(* Logix 5000 project; controller LeakTestAuto vendor 1 type 14 code 226 rev 37.11; software revision 37.01; part 7 of 15 *)
(* tags used below, declared in another part *)
   ConveyorPurgeCounter : DINT;   // Outfeed Coveyor Purge Counter
   DateString : String20;
   DateTimeString : String20;
   HMI_PurgeCycleSP : DINT;   // HMI Purge Cycles Setpoint
   I_OP220_N3_CONVEYOR_CLEAT : ALIAS FOR Local:3:I.Pt13.Data;
   I_OP220_N3_CONVEYOR_LOAD : ALIAS FOR Local:3:I.Pt12.Data;
   I_OP220_N3_CONVEYOR_UNLOAD : ALIAS FOR Local:3:I.Pt14.Data;
   I_OP220_N3_DUT_PRE_NEST_0 : ALIAS FOR Local:3:I.Pt00.Data;
   I_OP220_N3_DUT_PRE_NEST_1 : ALIAS FOR Local:3:I.Pt01.Data;
   I_OP220_N3_DUT_PRE_NEST_2 : ALIAS FOR Local:3:I.Pt02.Data;
   I_OP220_N3_MAIN_AIR_OK : ALIAS FOR Local:3:I.Pt07.Data;
   I_OP220_N3_NEST1_EXTEND : ALIAS FOR Local:3:I.Pt04.Data;
   I_OP220_N3_NEST1_HOME : ALIAS FOR Local:3:I.Pt03.Data;
   I_OP220_N3_NEST2_EXTEND : ALIAS FOR Local:3:I.Pt06.Data;
   I_OP220_N3_NEST2_HOME : ALIAS FOR Local:3:I.Pt05.Data;
   I_OP220_N3_REJECT_BIN_OK : ALIAS FOR Local:3:I.Pt09.Data;
   IOCounterHasRef : BOOL;
   IOTriggerCounts : UDINT[128];
   James_Dint : DINT;   // James Test Word
   LastPLCEdit : String20;
   LastPLCEditHistory : String20[20];
   O_OP220_N5_EN_LT_BU : ALIAS FOR Local:5:O.Pt03.Data;
   O_OP220_N5_EN_LT_GN : ALIAS FOR Local:5:O.Pt00.Data;
   O_OP220_N5_EN_LT_RD : ALIAS FOR Local:5:O.Pt02.Data;
   O_OP220_N5_EN_LT_YE : ALIAS FOR Local:5:O.Pt01.Data;
   OP220_ConsumedFromMain_PurgeModeEn : BOOL;
   OP220_Power : BOOL;
   PLC : AOI_PLC;
   Purge_Count_DN : BOOL;   // Purge Counter Completed
   ShiftChange : BOOL;
   ShiftNumber : SINT;
   TimeString : String20;
   TON_PLC_BootUp : TIMER;

        [95].VolumeTest.Detailed.Test_Type := 69, [95].VolumeTest.Detailed.element_data[0].Variable_code := 245, [95].VolumeTest.Detailed.element_data[0].prec_code := 2, [95].VolumeTest.Detailed.element_data[0].Unit_code := 165, [95].VolumeTest.Detailed.element_data[0].result_measurement := 188.38309, [95].VolumeTest.Detailed.element_data[1].Variable_code := 13, [95].VolumeTest.Detailed.element_data[1].prec_code := 3, [95].VolumeTest.Detailed.element_data[1].Unit_code := 12, [95].VolumeTest.Detailed.element_data[1].result_measurement := 1.8068217, [95].VolumeTest.Detailed.element_data[2].Variable_code := 247, [95].VolumeTest.Detailed.element_data[2].prec_code := 3, [95].VolumeTest.Detailed.element_data[2].Unit_code := 12, [95].VolumeTest.Detailed.element_data[2].result_measurement := 5.2105684, [95].VolumeTest.Detailed.element_data[3].Variable_code := 295, [95].VolumeTest.Detailed.element_data[3].prec_code := 3, [95].VolumeTest.Detailed.element_data[3].Unit_code := 12, [95].VolumeTest.Detailed.element_data[3].result_measurement := 5.212333, [95].LeakTest.UID := 42962, [95].LeakTest.Basic.unique_id := 42962, [95].LeakTest.Basic.channel_num := 1, [95].LeakTest.Basic.program_num := 2, [95].LeakTest.Basic.evaluation_code := 1, [95].LeakTest.Basic.test_port := 1, [95].LeakTest.Basic.year := 26, [95].LeakTest.Basic.month := 6, [95].LeakTest.Basic.date := 4, [95].LeakTest.Basic.hour := 15, [95].LeakTest.Basic.minute := 9, [95].LeakTest.Basic.second := 47, [95].LeakTest.Basic.flags := 12, [95].LeakTest.Basic.Num_tests := 1, [95].LeakTest.Basic.test_elements.test_type := 66, [95].LeakTest.Basic.test_elements.test_eval := 1, [95].LeakTest.Basic.test_elements.num_elements := 16, [95].LeakTest.Detailed.unique_id := 42962, [95].LeakTest.Detailed.num_elements := 16, [95].LeakTest.Detailed.Test_Type := 66, [95].LeakTest.Detailed.element_data[0].Variable_code := 61, [95].LeakTest.Detailed.element_data[0].prec_code := 2, [95].LeakTest.Detailed.element_data[0].Unit_code := 60, [95].LeakTest.Detailed.element_data[0].result_measurement := 0.022351742, [95].LeakTest.Detailed.element_data[1].Variable_code := 28, [95].LeakTest.Detailed.element_data[1].prec_code := 3, [95].LeakTest.Detailed.element_data[1].Unit_code := 41, [95].LeakTest.Detailed.element_data[1].result_measurement := 0.0004656613, [95].LeakTest.Detailed.element_data[2].Variable_code := 13, [95].LeakTest.Detailed.element_data[2].prec_code := 3, [95].LeakTest.Detailed.element_data[2].Unit_code := 12, [95].LeakTest.Detailed.element_data[2].result_measurement := 5.2300653, [95].LeakTest.Detailed.element_data[3].Variable_code := 75, [95].LeakTest.Detailed.element_data[3].prec_code := 2, [95].LeakTest.Detailed.element_data[3].Unit_code := 60, [95].LeakTest.Detailed.element_data[4].Variable_code := 60, [95].LeakTest.Detailed.element_data[4].prec_code := 2, [95].LeakTest.Detailed.element_data[4].Unit_code := 60, [95].LeakTest.Detailed.element_data[4].result_measurement := 0.022910535, [95].LeakTest.Detailed.element_data[5].Variable_code := 56, [95].LeakTest.Detailed.element_data[5].prec_code := 3, [95].LeakTest.Detailed.element_data[5].Unit_code := 41, [95].LeakTest.Detailed.element_data[5].result_measurement := 0.00020023435,
        [95].LeakTest.Detailed.element_data[6].Variable_code := 55, [95].LeakTest.Detailed.element_data[6].prec_code := 3, [95].LeakTest.Detailed.element_data[6].Unit_code := 12, [95].LeakTest.Detailed.element_data[6].result_measurement := 5.2300653, [95].LeakTest.Detailed.element_data[7].Variable_code := 58, [95].LeakTest.Detailed.element_data[7].prec_code := 2, [95].LeakTest.Detailed.element_data[7].Unit_code := 60, [95].LeakTest.Detailed.element_data[7].result_measurement := -1.0002404, [95].LeakTest.Detailed.element_data[8].Variable_code := 59, [95].LeakTest.Detailed.element_data[8].prec_code := 2, [95].LeakTest.Detailed.element_data[8].Unit_code := 60, [95].LeakTest.Detailed.element_data[8].result_measurement := 1.0002404, [95].LeakTest.Detailed.element_data[9].Variable_code := 12, [95].LeakTest.Detailed.element_data[9].prec_code := 3, [95].LeakTest.Detailed.element_data[9].Unit_code := 12, [95].LeakTest.Detailed.element_data[9].result_measurement := 5.000001, [95].LeakTest.Detailed.element_data[10].Variable_code := 62, [95].LeakTest.Detailed.element_data[10].prec_code := 2, [95].LeakTest.Detailed.element_data[10].Unit_code := 60, [95].LeakTest.Detailed.element_data[10].result_measurement := 1.1298805, [95].LeakTest.Detailed.element_data[11].Variable_code := 21, [95].LeakTest.Detailed.element_data[11].prec_code := 3, [95].LeakTest.Detailed.element_data[11].Unit_code := 41, [95].LeakTest.Detailed.element_data[11].result_measurement := 4.656613e-06, [95].LeakTest.Detailed.element_data[12].Variable_code := 25, [95].LeakTest.Detailed.element_data[12].prec_code := 3, [95].LeakTest.Detailed.element_data[12].Unit_code := 41, [95].LeakTest.Detailed.element_data[12].result_measurement := 0.023245811, [95].LeakTest.Detailed.element_data[13].Variable_code := 216, [95].LeakTest.Detailed.element_data[13].prec_code := 3, [95].LeakTest.Detailed.element_data[13].Unit_code := 41, [95].LeakTest.Detailed.element_data[13].result_measurement := -3.7252903e-05, [95].LeakTest.Detailed.element_data[14].Variable_code := 218, [95].LeakTest.Detailed.element_data[14].prec_code := 3, [95].LeakTest.Detailed.element_data[14].Unit_code := 41, [95].LeakTest.Detailed.element_data[14].result_measurement := 0.011632219, [95].LeakTest.Detailed.element_data[15].Variable_code := 295, [95].LeakTest.Detailed.element_data[15].prec_code := 3, [95].LeakTest.Detailed.element_data[15].Unit_code := 12, [95].LeakTest.Detailed.element_data[15].result_measurement := 5.231574, [96].Barcode := 'B252620865', [96].VolumeTest.UID := 42009, [96].VolumeTest.Basic.unique_id := 42009, [96].VolumeTest.Basic.channel_num := 1, [96].VolumeTest.Basic.program_num := 1, [96].VolumeTest.Basic.evaluation_code := 1, [96].VolumeTest.Basic.test_port := 1, [96].VolumeTest.Basic.year := 26, [96].VolumeTest.Basic.month := 6, [96].VolumeTest.Basic.date := 5, [96].VolumeTest.Basic.hour := 10, [96].VolumeTest.Basic.minute := 13, [96].VolumeTest.Basic.second := 35, [96].VolumeTest.Basic.flags := 12, [96].VolumeTest.Basic.Num_tests := 1, [96].VolumeTest.Basic.test_elements.test_type := 69, [96].VolumeTest.Basic.test_elements.test_eval := 1, [96].VolumeTest.Basic.test_elements.num_elements := 4, [96].VolumeTest.Detailed.unique_id := 42009, [96].VolumeTest.Detailed.num_elements := 4,
        [96].VolumeTest.Detailed.Test_Type := 69, [96].VolumeTest.Detailed.element_data[0].Variable_code := 245, [96].VolumeTest.Detailed.element_data[0].prec_code := 2, [96].VolumeTest.Detailed.element_data[0].Unit_code := 165, [96].VolumeTest.Detailed.element_data[0].result_measurement := 185.74803, [96].VolumeTest.Detailed.element_data[1].Variable_code := 13, [96].VolumeTest.Detailed.element_data[1].prec_code := 3, [96].VolumeTest.Detailed.element_data[1].Unit_code := 12, [96].VolumeTest.Detailed.element_data[1].result_measurement := 1.7781556, [96].VolumeTest.Detailed.element_data[2].Variable_code := 247, [96].VolumeTest.Detailed.element_data[2].prec_code := 3, [96].VolumeTest.Detailed.element_data[2].Unit_code := 12, [96].VolumeTest.Detailed.element_data[2].result_measurement := 5.0810447, [96].VolumeTest.Detailed.element_data[3].Variable_code := 295, [96].VolumeTest.Detailed.element_data[3].prec_code := 3, [96].VolumeTest.Detailed.element_data[3].Unit_code := 12, [96].VolumeTest.Detailed.element_data[3].result_measurement := 5.081105, [96].LeakTest.UID := 42010, [96].LeakTest.Basic.unique_id := 42010, [96].LeakTest.Basic.channel_num := 1, [96].LeakTest.Basic.program_num := 2, [96].LeakTest.Basic.evaluation_code := 1, [96].LeakTest.Basic.test_port := 1, [96].LeakTest.Basic.year := 26, [96].LeakTest.Basic.month := 6, [96].LeakTest.Basic.date := 5, [96].LeakTest.Basic.hour := 10, [96].LeakTest.Basic.minute := 13, [96].LeakTest.Basic.second := 42, [96].LeakTest.Basic.flags := 12, [96].LeakTest.Basic.Num_tests := 1, [96].LeakTest.Basic.test_elements.test_type := 66, [96].LeakTest.Basic.test_elements.test_eval := 1, [96].LeakTest.Basic.test_elements.num_elements := 16, [96].LeakTest.Detailed.unique_id := 42010, [96].LeakTest.Detailed.num_elements := 16, [96].LeakTest.Detailed.Test_Type := 66, [96].LeakTest.Detailed.element_data[0].Variable_code := 61, [96].LeakTest.Detailed.element_data[0].prec_code := 2, [96].LeakTest.Detailed.element_data[0].Unit_code := 60, [96].LeakTest.Detailed.element_data[0].result_measurement := -0.067055225, [96].LeakTest.Detailed.element_data[1].Variable_code := 28, [96].LeakTest.Detailed.element_data[1].prec_code := 3, [96].LeakTest.Detailed.element_data[1].Unit_code := 41, [96].LeakTest.Detailed.element_data[1].result_measurement := 0.00027939677, [96].LeakTest.Detailed.element_data[2].Variable_code := 13, [96].LeakTest.Detailed.element_data[2].prec_code := 3, [96].LeakTest.Detailed.element_data[2].Unit_code := 12, [96].LeakTest.Detailed.element_data[2].result_measurement := 5.1023254, [96].LeakTest.Detailed.element_data[3].Variable_code := 75, [96].LeakTest.Detailed.element_data[3].prec_code := 2, [96].LeakTest.Detailed.element_data[3].Unit_code := 60, [96].LeakTest.Detailed.element_data[4].Variable_code := 60, [96].LeakTest.Detailed.element_data[4].prec_code := 2, [96].LeakTest.Detailed.element_data[4].Unit_code := 60, [96].LeakTest.Detailed.element_data[4].result_measurement := -0.07208437, [96].LeakTest.Detailed.element_data[5].Variable_code := 56, [96].LeakTest.Detailed.element_data[5].prec_code := 3, [96].LeakTest.Detailed.element_data[5].Unit_code := 41, [96].LeakTest.Detailed.element_data[5].result_measurement := 0.00019092113,
        [96].LeakTest.Detailed.element_data[6].Variable_code := 55, [96].LeakTest.Detailed.element_data[6].prec_code := 3, [96].LeakTest.Detailed.element_data[6].Unit_code := 12, [96].LeakTest.Detailed.element_data[6].result_measurement := 5.1023254, [96].LeakTest.Detailed.element_data[7].Variable_code := 58, [96].LeakTest.Detailed.element_data[7].prec_code := 2, [96].LeakTest.Detailed.element_data[7].Unit_code := 60, [96].LeakTest.Detailed.element_data[7].result_measurement := -1.0002404, [96].LeakTest.Detailed.element_data[8].Variable_code := 59, [96].LeakTest.Detailed.element_data[8].prec_code := 2, [96].LeakTest.Detailed.element_data[8].Unit_code := 60, [96].LeakTest.Detailed.element_data[8].result_measurement := 1.0002404, [96].LeakTest.Detailed.element_data[9].Variable_code := 12, [96].LeakTest.Detailed.element_data[9].prec_code := 3, [96].LeakTest.Detailed.element_data[9].Unit_code := 12, [96].LeakTest.Detailed.element_data[9].result_measurement := 5.000001, [96].LeakTest.Detailed.element_data[10].Variable_code := 62, [96].LeakTest.Detailed.element_data[10].prec_code := 2, [96].LeakTest.Detailed.element_data[10].Unit_code := 60, [96].LeakTest.Detailed.element_data[10].result_measurement := 1.1002644, [96].LeakTest.Detailed.element_data[11].Variable_code := 21, [96].LeakTest.Detailed.element_data[11].prec_code := 3, [96].LeakTest.Detailed.element_data[11].Unit_code := 41, [96].LeakTest.Detailed.element_data[11].result_measurement := 0.0015180558, [96].LeakTest.Detailed.element_data[12].Variable_code := 25, [96].LeakTest.Detailed.element_data[12].prec_code := 3, [96].LeakTest.Detailed.element_data[12].Unit_code := 41, [96].LeakTest.Detailed.element_data[12].result_measurement := 0.021727756, [96].LeakTest.Detailed.element_data[13].Variable_code := 216, [96].LeakTest.Detailed.element_data[13].prec_code := 3, [96].LeakTest.Detailed.element_data[13].Unit_code := 41, [96].LeakTest.Detailed.element_data[13].result_measurement := 0.00085681677, [96].LeakTest.Detailed.element_data[14].Variable_code := 218, [96].LeakTest.Detailed.element_data[14].prec_code := 3, [96].LeakTest.Detailed.element_data[14].Unit_code := 41, [96].LeakTest.Detailed.element_data[14].result_measurement := 0.01094304, [96].LeakTest.Detailed.element_data[15].Variable_code := 295, [96].LeakTest.Detailed.element_data[15].prec_code := 3, [96].LeakTest.Detailed.element_data[15].Unit_code := 12, [96].LeakTest.Detailed.element_data[15].result_measurement := 5.1039925, [97].Barcode := 'B252620970', [97].VolumeTest.UID := 42015, [97].VolumeTest.Basic.unique_id := 42015, [97].VolumeTest.Basic.channel_num := 1, [97].VolumeTest.Basic.program_num := 1, [97].VolumeTest.Basic.evaluation_code := 1, [97].VolumeTest.Basic.test_port := 1, [97].VolumeTest.Basic.year := 26, [97].VolumeTest.Basic.month := 6, [97].VolumeTest.Basic.date := 5, [97].VolumeTest.Basic.hour := 10, [97].VolumeTest.Basic.minute := 18, [97].VolumeTest.Basic.second := 26, [97].VolumeTest.Basic.flags := 12, [97].VolumeTest.Basic.Num_tests := 1, [97].VolumeTest.Basic.test_elements.test_type := 69, [97].VolumeTest.Basic.test_elements.test_eval := 1, [97].VolumeTest.Basic.test_elements.num_elements := 4, [97].VolumeTest.Detailed.unique_id := 42015, [97].VolumeTest.Detailed.num_elements := 4,
        [97].VolumeTest.Detailed.Test_Type := 69, [97].VolumeTest.Detailed.element_data[0].Variable_code := 245, [97].VolumeTest.Detailed.element_data[0].prec_code := 2, [97].VolumeTest.Detailed.element_data[0].Unit_code := 165, [97].VolumeTest.Detailed.element_data[0].result_measurement := 185.95625, [97].VolumeTest.Detailed.element_data[1].Variable_code := 13, [97].VolumeTest.Detailed.element_data[1].prec_code := 3, [97].VolumeTest.Detailed.element_data[1].Unit_code := 12, [97].VolumeTest.Detailed.element_data[1].result_measurement := 1.778258, [97].VolumeTest.Detailed.element_data[2].Variable_code := 247, [97].VolumeTest.Detailed.element_data[2].prec_code := 3, [97].VolumeTest.Detailed.element_data[2].Unit_code := 12, [97].VolumeTest.Detailed.element_data[2].result_measurement := 5.08504, [97].VolumeTest.Detailed.element_data[3].Variable_code := 295, [97].VolumeTest.Detailed.element_data[3].prec_code := 3, [97].VolumeTest.Detailed.element_data[3].Unit_code := 12, [97].VolumeTest.Detailed.element_data[3].result_measurement := 5.086218, [97].LeakTest.UID := 42016, [97].LeakTest.Basic.unique_id := 42016, [97].LeakTest.Basic.channel_num := 1, [97].LeakTest.Basic.program_num := 2, [97].LeakTest.Basic.evaluation_code := 1, [97].LeakTest.Basic.test_port := 1, [97].LeakTest.Basic.year := 26, [97].LeakTest.Basic.month := 6, [97].LeakTest.Basic.date := 5, [97].LeakTest.Basic.hour := 10, [97].LeakTest.Basic.minute := 18, [97].LeakTest.Basic.second := 33, [97].LeakTest.Basic.flags := 12, [97].LeakTest.Basic.Num_tests := 1, [97].LeakTest.Basic.test_elements.test_type := 66, [97].LeakTest.Basic.test_elements.test_eval := 1, [97].LeakTest.Basic.test_elements.num_elements := 16, [97].LeakTest.Detailed.unique_id := 42016, [97].LeakTest.Detailed.num_elements := 16, [97].LeakTest.Detailed.Test_Type := 66, [97].LeakTest.Detailed.element_data[0].Variable_code := 61, [97].LeakTest.Detailed.element_data[0].prec_code := 2, [97].LeakTest.Detailed.element_data[0].Unit_code := 60, [97].LeakTest.Detailed.element_data[0].result_measurement := -0.0692904, [97].LeakTest.Detailed.element_data[1].Variable_code := 28, [97].LeakTest.Detailed.element_data[1].prec_code := 3, [97].LeakTest.Detailed.element_data[1].Unit_code := 41, [97].LeakTest.Detailed.element_data[1].result_measurement := 0.00023748726, [97].LeakTest.Detailed.element_data[2].Variable_code := 13, [97].LeakTest.Detailed.element_data[2].prec_code := 3, [97].LeakTest.Detailed.element_data[2].Unit_code := 12, [97].LeakTest.Detailed.element_data[2].result_measurement := 5.1036057, [97].LeakTest.Detailed.element_data[3].Variable_code := 75, [97].LeakTest.Detailed.element_data[3].prec_code := 2, [97].LeakTest.Detailed.element_data[3].Unit_code := 60, [97].LeakTest.Detailed.element_data[4].Variable_code := 60, [97].LeakTest.Detailed.element_data[4].prec_code := 2, [97].LeakTest.Detailed.element_data[4].Unit_code := 60, [97].LeakTest.Detailed.element_data[4].result_measurement := -0.073201954, [97].LeakTest.Detailed.element_data[5].Variable_code := 56, [97].LeakTest.Detailed.element_data[5].prec_code := 3, [97].LeakTest.Detailed.element_data[5].Unit_code := 41, [97].LeakTest.Detailed.element_data[5].result_measurement := 0.0001816079,
        [97].LeakTest.Detailed.element_data[6].Variable_code := 55, [97].LeakTest.Detailed.element_data[6].prec_code := 3, [97].LeakTest.Detailed.element_data[6].Unit_code := 12, [97].LeakTest.Detailed.element_data[6].result_measurement := 5.1036057, [97].LeakTest.Detailed.element_data[7].Variable_code := 58, [97].LeakTest.Detailed.element_data[7].prec_code := 2, [97].LeakTest.Detailed.element_data[7].Unit_code := 60, [97].LeakTest.Detailed.element_data[7].result_measurement := -1.0002404, [97].LeakTest.Detailed.element_data[8].Variable_code := 59, [97].LeakTest.Detailed.element_data[8].prec_code := 2, [97].LeakTest.Detailed.element_data[8].Unit_code := 60, [97].LeakTest.Detailed.element_data[8].result_measurement := 1.0002404, [97].LeakTest.Detailed.element_data[9].Variable_code := 12, [97].LeakTest.Detailed.element_data[9].prec_code := 3, [97].LeakTest.Detailed.element_data[9].Unit_code := 12, [97].LeakTest.Detailed.element_data[9].result_measurement := 5.000001, [97].LeakTest.Detailed.element_data[10].Variable_code := 62, [97].LeakTest.Detailed.element_data[10].prec_code := 2, [97].LeakTest.Detailed.element_data[10].Unit_code := 60, [97].LeakTest.Detailed.element_data[10].result_measurement := 1.1002644, [97].LeakTest.Detailed.element_data[11].Variable_code := 21, [97].LeakTest.Detailed.element_data[11].prec_code := 3, [97].LeakTest.Detailed.element_data[11].Unit_code := 41, [97].LeakTest.Detailed.element_data[11].result_measurement := 0.0015180558, [97].LeakTest.Detailed.element_data[12].Variable_code := 25, [97].LeakTest.Detailed.element_data[12].prec_code := 3, [97].LeakTest.Detailed.element_data[12].Unit_code := 41, [97].LeakTest.Detailed.element_data[12].result_measurement := 0.021727756, [97].LeakTest.Detailed.element_data[13].Variable_code := 216, [97].LeakTest.Detailed.element_data[13].prec_code := 3, [97].LeakTest.Detailed.element_data[13].Unit_code := 41, [97].LeakTest.Detailed.element_data[13].result_measurement := 0.00085681677, [97].LeakTest.Detailed.element_data[14].Variable_code := 218, [97].LeakTest.Detailed.element_data[14].prec_code := 3, [97].LeakTest.Detailed.element_data[14].Unit_code := 41, [97].LeakTest.Detailed.element_data[14].result_measurement := 0.01094304, [97].LeakTest.Detailed.element_data[15].Variable_code := 295, [97].LeakTest.Detailed.element_data[15].prec_code := 3, [97].LeakTest.Detailed.element_data[15].Unit_code := 12, [97].LeakTest.Detailed.element_data[15].result_measurement := 5.1049933, [98].Barcode := 'B252620571', [98].VolumeTest.UID := 43010, [98].VolumeTest.Basic.unique_id := 43010, [98].VolumeTest.Basic.channel_num := 1, [98].VolumeTest.Basic.program_num := 1, [98].VolumeTest.Basic.evaluation_code := 1, [98].VolumeTest.Basic.test_port := 1, [98].VolumeTest.Basic.year := 26, [98].VolumeTest.Basic.month := 6, [98].VolumeTest.Basic.date := 5, [98].VolumeTest.Basic.hour := 10, [98].VolumeTest.Basic.minute := 18, [98].VolumeTest.Basic.second := 50, [98].VolumeTest.Basic.flags := 12, [98].VolumeTest.Basic.Num_tests := 1, [98].VolumeTest.Basic.test_elements.test_type := 69, [98].VolumeTest.Basic.test_elements.test_eval := 1, [98].VolumeTest.Basic.test_elements.num_elements := 4, [98].VolumeTest.Detailed.unique_id := 43010, [98].VolumeTest.Detailed.num_elements := 4,
        [98].VolumeTest.Detailed.Test_Type := 69, [98].VolumeTest.Detailed.element_data[0].Variable_code := 245, [98].VolumeTest.Detailed.element_data[0].prec_code := 2, [98].VolumeTest.Detailed.element_data[0].Unit_code := 165, [98].VolumeTest.Detailed.element_data[0].result_measurement := 187.18771, [98].VolumeTest.Detailed.element_data[1].Variable_code := 13, [98].VolumeTest.Detailed.element_data[1].prec_code := 3, [98].VolumeTest.Detailed.element_data[1].Unit_code := 12, [98].VolumeTest.Detailed.element_data[1].result_measurement := 1.7792639, [98].VolumeTest.Detailed.element_data[2].Variable_code := 247, [98].VolumeTest.Detailed.element_data[2].prec_code := 3, [98].VolumeTest.Detailed.element_data[2].Unit_code := 12, [98].VolumeTest.Detailed.element_data[2].result_measurement := 5.109827, [98].VolumeTest.Detailed.element_data[3].Variable_code := 295, [98].VolumeTest.Detailed.element_data[3].prec_code := 3, [98].VolumeTest.Detailed.element_data[3].Unit_code := 12, [98].VolumeTest.Detailed.element_data[3].result_measurement := 5.1112704, [98].LeakTest.UID := 43011, [98].LeakTest.Basic.unique_id := 43011, [98].LeakTest.Basic.channel_num := 1, [98].LeakTest.Basic.program_num := 2, [98].LeakTest.Basic.evaluation_code := 1, [98].LeakTest.Basic.test_port := 1, [98].LeakTest.Basic.year := 26, [98].LeakTest.Basic.month := 6, [98].LeakTest.Basic.date := 5, [98].LeakTest.Basic.hour := 10, [98].LeakTest.Basic.minute := 18, [98].LeakTest.Basic.second := 57, [98].LeakTest.Basic.flags := 12, [98].LeakTest.Basic.Num_tests := 1, [98].LeakTest.Basic.test_elements.test_type := 66, [98].LeakTest.Basic.test_elements.test_eval := 1, [98].LeakTest.Basic.test_elements.num_elements := 16, [98].LeakTest.Detailed.unique_id := 43011, [98].LeakTest.Detailed.num_elements := 16, [98].LeakTest.Detailed.Test_Type := 66, [98].LeakTest.Detailed.element_data[0].Variable_code := 61, [98].LeakTest.Detailed.element_data[0].prec_code := 2, [98].LeakTest.Detailed.element_data[0].Unit_code := 60, [98].LeakTest.Detailed.element_data[0].result_measurement := -0.0033527613, [98].LeakTest.Detailed.element_data[1].Variable_code := 28, [98].LeakTest.Detailed.element_data[1].prec_code := 3, [98].LeakTest.Detailed.element_data[1].Unit_code := 41, [98].LeakTest.Detailed.element_data[1].result_measurement := -7.4505806e-05, [98].LeakTest.Detailed.element_data[2].Variable_code := 13, [98].LeakTest.Detailed.element_data[2].prec_code := 3, [98].LeakTest.Detailed.element_data[2].Unit_code := 12, [98].LeakTest.Detailed.element_data[2].result_measurement := 5.146088, [98].LeakTest.Detailed.element_data[3].Variable_code := 75, [98].LeakTest.Detailed.element_data[3].prec_code := 2, [98].LeakTest.Detailed.element_data[3].Unit_code := 60, [98].LeakTest.Detailed.element_data[4].Variable_code := 60, [98].LeakTest.Detailed.element_data[4].prec_code := 2, [98].LeakTest.Detailed.element_data[4].Unit_code := 60, [98].LeakTest.Detailed.element_data[4].result_measurement := 0.007264316, [98].LeakTest.Detailed.element_data[5].Variable_code := 56, [98].LeakTest.Detailed.element_data[5].prec_code := 3, [98].LeakTest.Detailed.element_data[5].Unit_code := 41, [98].LeakTest.Detailed.element_data[5].result_measurement := 4.1909516e-05,
        [98].LeakTest.Detailed.element_data[6].Variable_code := 55, [98].LeakTest.Detailed.element_data[6].prec_code := 3, [98].LeakTest.Detailed.element_data[6].Unit_code := 12, [98].LeakTest.Detailed.element_data[6].result_measurement := 5.146088, [98].LeakTest.Detailed.element_data[7].Variable_code := 58, [98].LeakTest.Detailed.element_data[7].prec_code := 2, [98].LeakTest.Detailed.element_data[7].Unit_code := 60, [98].LeakTest.Detailed.element_data[7].result_measurement := -1.0002404, [98].LeakTest.Detailed.element_data[8].Variable_code := 59, [98].LeakTest.Detailed.element_data[8].prec_code := 2, [98].LeakTest.Detailed.element_data[8].Unit_code := 60, [98].LeakTest.Detailed.element_data[8].result_measurement := 1.0002404, [98].LeakTest.Detailed.element_data[9].Variable_code := 12, [98].LeakTest.Detailed.element_data[9].prec_code := 3, [98].LeakTest.Detailed.element_data[9].Unit_code := 12, [98].LeakTest.Detailed.element_data[9].result_measurement := 5.000001, [98].LeakTest.Detailed.element_data[10].Variable_code := 62, [98].LeakTest.Detailed.element_data[10].prec_code := 2, [98].LeakTest.Detailed.element_data[10].Unit_code := 60, [98].LeakTest.Detailed.element_data[10].result_measurement := 1.1298805, [98].LeakTest.Detailed.element_data[11].Variable_code := 21, [98].LeakTest.Detailed.element_data[11].prec_code := 3, [98].LeakTest.Detailed.element_data[11].Unit_code := 41, [98].LeakTest.Detailed.element_data[11].result_measurement := 4.656613e-06, [98].LeakTest.Detailed.element_data[12].Variable_code := 25, [98].LeakTest.Detailed.element_data[12].prec_code := 3, [98].LeakTest.Detailed.element_data[12].Unit_code := 41, [98].LeakTest.Detailed.element_data[12].result_measurement := 0.023245811, [98].LeakTest.Detailed.element_data[13].Variable_code := 216, [98].LeakTest.Detailed.element_data[13].prec_code := 3, [98].LeakTest.Detailed.element_data[13].Unit_code := 41, [98].LeakTest.Detailed.element_data[13].result_measurement := -3.7252903e-05, [98].LeakTest.Detailed.element_data[14].Variable_code := 218, [98].LeakTest.Detailed.element_data[14].prec_code := 3, [98].LeakTest.Detailed.element_data[14].Unit_code := 41, [98].LeakTest.Detailed.element_data[14].result_measurement := 0.011632219, [98].LeakTest.Detailed.element_data[15].Variable_code := 295, [98].LeakTest.Detailed.element_data[15].prec_code := 3, [98].LeakTest.Detailed.element_data[15].Unit_code := 12, [98].LeakTest.Detailed.element_data[15].result_measurement := 5.147038, [99].Barcode := 'B252620863', [99].VolumeTest.UID := 43013, [99].VolumeTest.Basic.unique_id := 43013, [99].VolumeTest.Basic.channel_num := 1, [99].VolumeTest.Basic.program_num := 1, [99].VolumeTest.Basic.evaluation_code := 1, [99].VolumeTest.Basic.test_port := 1, [99].VolumeTest.Basic.year := 26, [99].VolumeTest.Basic.month := 6, [99].VolumeTest.Basic.date := 5, [99].VolumeTest.Basic.hour := 10, [99].VolumeTest.Basic.minute := 19, [99].VolumeTest.Basic.second := 44, [99].VolumeTest.Basic.flags := 12, [99].VolumeTest.Basic.Num_tests := 1, [99].VolumeTest.Basic.test_elements.test_type := 69, [99].VolumeTest.Basic.test_elements.test_eval := 1, [99].VolumeTest.Basic.test_elements.num_elements := 4, [99].VolumeTest.Detailed.unique_id := 43013, [99].VolumeTest.Detailed.num_elements := 4,
        [99].VolumeTest.Detailed.Test_Type := 69, [99].VolumeTest.Detailed.element_data[0].Variable_code := 245, [99].VolumeTest.Detailed.element_data[0].prec_code := 2, [99].VolumeTest.Detailed.element_data[0].Unit_code := 165, [99].VolumeTest.Detailed.element_data[0].result_measurement := 187.24707, [99].VolumeTest.Detailed.element_data[1].Variable_code := 13, [99].VolumeTest.Detailed.element_data[1].prec_code := 3, [99].VolumeTest.Detailed.element_data[1].Unit_code := 12, [99].VolumeTest.Detailed.element_data[1].result_measurement := 1.7789285, [99].VolumeTest.Detailed.element_data[2].Variable_code := 247, [99].VolumeTest.Detailed.element_data[2].prec_code := 3, [99].VolumeTest.Detailed.element_data[2].Unit_code := 12, [99].VolumeTest.Detailed.element_data[2].result_measurement := 5.10992, [99].VolumeTest.Detailed.element_data[3].Variable_code := 295, [99].VolumeTest.Detailed.element_data[3].prec_code := 3, [99].VolumeTest.Detailed.element_data[3].Unit_code := 12, [99].VolumeTest.Detailed.element_data[3].result_measurement := 5.111359, [99].LeakTest.UID := 43014, [99].LeakTest.Basic.unique_id := 43014, [99].LeakTest.Basic.channel_num := 1, [99].LeakTest.Basic.program_num := 2, [99].LeakTest.Basic.evaluation_code := 1, [99].LeakTest.Basic.test_port := 1, [99].LeakTest.Basic.year := 26, [99].LeakTest.Basic.month := 6, [99].LeakTest.Basic.date := 5, [99].LeakTest.Basic.hour := 10, [99].LeakTest.Basic.minute := 19, [99].LeakTest.Basic.second := 51, [99].LeakTest.Basic.flags := 12, [99].LeakTest.Basic.Num_tests := 1, [99].LeakTest.Basic.test_elements.test_type := 66, [99].LeakTest.Basic.test_elements.test_eval := 1, [99].LeakTest.Basic.test_elements.num_elements := 16, [99].LeakTest.Detailed.unique_id := 43014, [99].LeakTest.Detailed.num_elements := 16, [99].LeakTest.Detailed.Test_Type := 66, [99].LeakTest.Detailed.element_data[0].Variable_code := 61, [99].LeakTest.Detailed.element_data[0].prec_code := 2, [99].LeakTest.Detailed.element_data[0].Unit_code := 60, [99].LeakTest.Detailed.element_data[0].result_measurement := 0.007264316, [99].LeakTest.Detailed.element_data[1].Variable_code := 28, [99].LeakTest.Detailed.element_data[1].prec_code := 3, [99].LeakTest.Detailed.element_data[1].Unit_code := 41, [99].LeakTest.Detailed.element_data[1].result_measurement := 0.00015832484, [99].LeakTest.Detailed.element_data[2].Variable_code := 13, [99].LeakTest.Detailed.element_data[2].prec_code := 3, [99].LeakTest.Detailed.element_data[2].Unit_code := 12, [99].LeakTest.Detailed.element_data[2].result_measurement := 5.146228, [99].LeakTest.Detailed.element_data[3].Variable_code := 75, [99].LeakTest.Detailed.element_data[3].prec_code := 2, [99].LeakTest.Detailed.element_data[3].Unit_code := 60, [99].LeakTest.Detailed.element_data[4].Variable_code := 60, [99].LeakTest.Detailed.element_data[4].prec_code := 2, [99].LeakTest.Detailed.element_data[4].Unit_code := 60, [99].LeakTest.Detailed.element_data[4].result_measurement := 0.014528632, [99].LeakTest.Detailed.element_data[5].Variable_code := 56, [99].LeakTest.Detailed.element_data[5].prec_code := 3, [99].LeakTest.Detailed.element_data[5].Unit_code := 41, [99].LeakTest.Detailed.element_data[5].result_measurement := 0.00011641532,
        [99].LeakTest.Detailed.element_data[6].Variable_code := 55, [99].LeakTest.Detailed.element_data[6].prec_code := 3, [99].LeakTest.Detailed.element_data[6].Unit_code := 12, [99].LeakTest.Detailed.element_data[6].result_measurement := 5.146228, [99].LeakTest.Detailed.element_data[7].Variable_code := 58, [99].LeakTest.Detailed.element_data[7].prec_code := 2, [99].LeakTest.Detailed.element_data[7].Unit_code := 60, [99].LeakTest.Detailed.element_data[7].result_measurement := -1.0002404, [99].LeakTest.Detailed.element_data[8].Variable_code := 59, [99].LeakTest.Detailed.element_data[8].prec_code := 2, [99].LeakTest.Detailed.element_data[8].Unit_code := 60, [99].LeakTest.Detailed.element_data[8].result_measurement := 1.0002404, [99].LeakTest.Detailed.element_data[9].Variable_code := 12, [99].LeakTest.Detailed.element_data[9].prec_code := 3, [99].LeakTest.Detailed.element_data[9].Unit_code := 12, [99].LeakTest.Detailed.element_data[9].result_measurement := 5.000001, [99].LeakTest.Detailed.element_data[10].Variable_code := 62, [99].LeakTest.Detailed.element_data[10].prec_code := 2, [99].LeakTest.Detailed.element_data[10].Unit_code := 60, [99].LeakTest.Detailed.element_data[10].result_measurement := 1.1298805, [99].LeakTest.Detailed.element_data[11].Variable_code := 21, [99].LeakTest.Detailed.element_data[11].prec_code := 3, [99].LeakTest.Detailed.element_data[11].Unit_code := 41, [99].LeakTest.Detailed.element_data[11].result_measurement := 4.656613e-06, [99].LeakTest.Detailed.element_data[12].Variable_code := 25, [99].LeakTest.Detailed.element_data[12].prec_code := 3, [99].LeakTest.Detailed.element_data[12].Unit_code := 41, [99].LeakTest.Detailed.element_data[12].result_measurement := 0.023245811, [99].LeakTest.Detailed.element_data[13].Variable_code := 216, [99].LeakTest.Detailed.element_data[13].prec_code := 3, [99].LeakTest.Detailed.element_data[13].Unit_code := 41, [99].LeakTest.Detailed.element_data[13].result_measurement := -3.7252903e-05, [99].LeakTest.Detailed.element_data[14].Variable_code := 218, [99].LeakTest.Detailed.element_data[14].prec_code := 3, [99].LeakTest.Detailed.element_data[14].Unit_code := 41, [99].LeakTest.Detailed.element_data[14].result_measurement := 0.011632219, [99].LeakTest.Detailed.element_data[15].Variable_code := 295, [99].LeakTest.Detailed.element_data[15].prec_code := 3, [99].LeakTest.Detailed.element_data[15].Unit_code := 12, [99].LeakTest.Detailed.element_data[15].result_measurement := 5.14742);
   EIPTemplateCommStatus : AOI_CommStatus;
   EIPTemplateDeviceInput : udt_EIPTemplateData;
   EIPTemplateDeviceOutput : udt_EIPTemplateData;
   EIPTemplateLocalInput : udt_EIPTemplateLocalInput;
   EIPTemplateLocalOutput : udt_EIPTemplateLocalOutput;
   FailCount : COUNTER := (PRE := 10);
   FaultsAndWarnings : STRING[96] := ([0] := 'Main power off', [1] := 'Main air not OK', [2] := 'EStop high', [3] := 'Guard doors open', [4] := 'Reject bin missing', [5] := 'No EIP connection to barcode scanner', [6] := 'No EIP connection to CTS1', [7] := 'No EIP connection to CTS2', [8] := 'No EIP connection to Robot', [9] := 'EStop Safety Block faulted', [10] := 'Barcode scanner fault', [11] := 'CTS1 fault', [12] := 'CTS2 fault', [13] := 'Robot fault', [14] := 'Robot gripper in unknown state', [15] := 'Conveyor alarm high', [16] := 'Cylinder 1 fault', [17] := 'Cylinder 2 fault', [18] := '24V DC not OK', [19] := 'Check conveyor cleat sensor', [32] := '3 in a row fault', [33] := '5 in an hour fault', [34] := '10 in a shift fault', [42] := 'Homing cycle overtime', [43] := 'Fail chute failed to register unit (Homing Seq)', [44] := 'Fail chute failed to register unit (Auto Seq)', [45] := 'Cylinder 1 down timeout', [46] := 'Cylinder 2 down timeout', [47] := 'Cylinder 1 up timeout', [48] := 'Cylinder 2 up timeout', [64] := 'Cycle stop requested', [65] := 'Cycle pause requested', [66] := 'Step mode active', [67] := 'Dry cycle active', [68] := 'MES bypass active', [74] := 'Main sequence stuck on step$0D$0A', [75] := 'Homing sequence stuck on step$0D$0A', [76] := 'CTS1 sequence stuck on step 9000', [77] := 'CTS2 sequence stuck on step 9000', [78] := 'Conveyor sequence stuck on step 9000', [79] := 'Main sequence stuck on step$0D$0A', [80] := 'Homing sequence stuck on step$0D$0A', [81] := 'CTS1 sequence stuck on step ', [82] := 'CTS2 sequence stuck on step ', [83] := 'Conveyor sequence stuck on step ', [84] := 'CTS1 test requested but interlock not met', [85] := 'CTS2 test requested but interlock not met', [86] := 'CTS1 not ready', [87] := 'CTS2 not ready', [88] := 'Robot movement requested but interlock not met', [89] := 'Conveyor movement requested but interlock not met', [90] := 'Nest 1 movement requested but interlock not met', [91] := 'Nest 2 movement requested but interlock not met', [94] := 'Fail bin full, please empty');
   FFLU_CTS1Leak : CONTROL := (LEN := 10, POS := 10, DN := 1);
   FFLU_CTS1Vol : CONTROL := (LEN := 10, POS := 10, DN := 1);
   FFLU_CTS2Leak : CONTROL := (LEN := 10, POS := 10, DN := 1);
   FFLU_CTS2Vol : CONTROL := (LEN := 10, POS := 10, DN := 1);
   FFLU_DUTHistory : CONTROL := (LEN := 100, POS := 100, DN := 1);
   FFLUDumpREAL : REAL;
   HMI_CloseDisplay : DINT := 12;
   HMI_OP220_ClearProcessFaultCounts_IND : BOOL;
   HMI_OP220_ClearProcessFaultCounts_PB : BOOL;
   HMI_TestPointer : DINT;
   HomingClearNestsBypass : BOOL := 1;
   InfeedCounter : COUNTER := (PRE := 9999999, ACC := 20);
   LastFaults : DINT[2] := ([0] := 205549);
   LastShiftNumber : DINT := 1;
   LeakTester1 : udt_OutputStructure := (REQ := 3);
   LeakTester2 : udt_OutputStructure := (REQ := 3);
   Mode_CapActuators : BOOL;
   Mode_CapCTS : BOOL;
   Mode_CapCylinders : BOOL;
   Mode_CapFail : BOOL;
   Mode_CapPass : BOOL;
   Mode_CapRobot : BOOL;
   Mode_CapShuffle : BOOL;
   Nest1Bypass : BOOL := 1;
   Nest1Cylinder : udt_OutputStructure := (BTMR.PRE := 500);
   Nest1Empty : BOOL := 1;
   Nest1Ready : BOOL;
   Nest2Bypass : BOOL := 1;
   Nest2Cylinder : udt_OutputStructure := (BTMR.PRE := 500);
   Nest2Empty : BOOL := 1;
   Nest2Ready : BOOL;
   ONS_AutoMode : BOOL := 1;
   ONS_CapActuators : BOOL;
   ONS_CapCTS : BOOL;
   ONS_CapCylinders : BOOL;
   ONS_CapFail : BOOL;
   ONS_CapPass : BOOL;
   ONS_CapRobot : BOOL;
   ONS_CapShuffle : BOOL;
   ONS_ClearWarnings : BOOL;
   ONS_CTS1ClearResultsBC : BOOL := 1;
   ONS_CTS1GetResults : BOOL;
   ONS_CTS1ResultHistory : BOOL;
   ONS_CTS2ClearResultsBC : BOOL := 1;
   ONS_CTS2GetResults : BOOL;
   ONS_CTS2ResultHistory : BOOL;
   ONS_CycleStop : BOOL;
   ONS_FailBinRemoved : BOOL;
   ONS_HMICloseDisplay : BOOL := 1;
   ONS_ManuMode : BOOL := 1;
   ONS_RobotGripper : SINT := 1;
   OP220 : udt_Mode := (PowerOn := 1, PowerOnONS := 1, AirOk := 1, UtilitiesOk := 1, EStopsOk := 1, GuardDoorsOk := 1, FaultActive := 1, WarningActive := 1, ReadyForAuto := 1, ManualMode := 1, Home := 1, MESBypass := 1, ManualMode_IND := 2, Home_IND := 2, HMIBackgroundIND := 2, Faults[0] := 205517, Faults[1] := 98304, Warnings[0] := 12582928, HomingOvertime.PRE := 120000, PowerOnTMR.PRE := 500, PowerOnTMR.ACC := 500, PowerOnTMR.EN := 1, PowerOnTMR.DN := 1, AirOKTMR.PRE := 500, AirOKTMR.ACC := 500, AirOKTMR.EN := 1, AirOKTMR.DN := 1, CycleStopOverideTMR.PRE := 3000, FaultTMR[0].TMR[0].PRE := 1, FaultTMR[0].TMR[1].PRE := 1, FaultTMR[0].TMR[2].PRE := 1, FaultTMR[0].TMR[3].PRE := 1, FaultTMR[0].TMR[4].PRE := 60000, FaultTMR[0].TMR[5].PRE := 1000, FaultTMR[0].TMR[5].ACC := 1000, FaultTMR[0].TMR[5].EN := 1, FaultTMR[0].TMR[5].DN := 1, FaultTMR[0].TMR[6].PRE := 1000, FaultTMR[0].TMR[6].ACC := 1000, FaultTMR[0].TMR[6].EN := 1, FaultTMR[0].TMR[6].DN := 1, FaultTMR[0].TMR[7].PRE := 1000, FaultTMR[0].TMR[7].ACC := 1000, FaultTMR[0].TMR[7].EN := 1, FaultTMR[0].TMR[7].DN := 1, FaultTMR[0].TMR[8].PRE := 1000, FaultTMR[0].TMR[9].PRE := 1, FaultTMR[0].TMR[10].PRE := 1, FaultTMR[0].TMR[11].PRE := 1, FaultTMR[0].TMR[12].PRE := 1, FaultTMR[0].TMR[13].PRE := 1, FaultTMR[0].TMR[14].PRE := 1, FaultTMR[0].TMR[15].PRE := 1000, FaultTMR[0].TMR[16].PRE := 1, FaultTMR[0].TMR[17].PRE := 1, FaultTMR[0].TMR[18].PRE := 1, FaultTMR[0].TMR[19].PRE := 1, FaultTMR[1].TMR[0].PRE := 1, FaultTMR[1].TMR[1].PRE := 1, FaultTMR[1].TMR[2].PRE := 1,
        FaultTMR[1].TMR[10].PRE := 1, FaultTMR[1].TMR[11].PRE := 1, FaultTMR[1].TMR[12].PRE := 1, FaultTMR[1].TMR[13].PRE := 1, FaultTMR[1].TMR[14].PRE := 1, FaultTMR[1].TMR[15].PRE := 1, FaultTMR[1].TMR[16].PRE := 1, FaultTMR[1].TMR[17].PRE := 1, FaultTMR[1].TMR[18].PRE := 1, FaultTMR[1].TMR[19].PRE := 1, FaultTMR[1].TMR[20].PRE := 1, WarningTMR[0].TMR[0].PRE := 1, WarningTMR[0].TMR[1].PRE := 1, WarningTMR[0].TMR[2].PRE := 1, WarningTMR[0].TMR[3].PRE := 1, WarningTMR[0].TMR[4].PRE := 1, WarningTMR[0].TMR[4].ACC := 1, WarningTMR[0].TMR[4].EN := 1, WarningTMR[0].TMR[4].DN := 1, WarningTMR[0].TMR[10].PRE := 1, WarningTMR[0].TMR[11].PRE := 1, WarningTMR[0].TMR[12].PRE := 1, WarningTMR[0].TMR[13].PRE := 1, WarningTMR[0].TMR[14].PRE := 1, WarningTMR[0].TMR[20].PRE := 2000, WarningTMR[0].TMR[21].PRE := 2000, WarningTMR[0].TMR[22].PRE := 30000, WarningTMR[0].TMR[22].ACC := 30000, WarningTMR[0].TMR[22].EN := 1, WarningTMR[0].TMR[22].DN := 1, WarningTMR[0].TMR[23].PRE := 30000, WarningTMR[0].TMR[23].ACC := 30000, WarningTMR[0].TMR[23].EN := 1, WarningTMR[0].TMR[23].DN := 1, WarningTMR[0].TMR[24].PRE := 5000, WarningTMR[0].TMR[25].PRE := 1000, WarningTMR[0].TMR[26].PRE := 1000, WarningTMR[0].TMR[27].PRE := 1000, WarningTMR[0].TMR[30].PRE := 1);
   OP220_Disable3510 : BOOL;
   OP220_Fault_Counter : COUNTER := (PRE := 9999999, ACC := 67);
   OP220_Fault_Counter_ONS : BOOL := 1;
   OP220_Fault_Number : DINT;
   OP220_Fault_Reset_ONS : BOOL;
   OP220_FaultCounter_Reset_ONS : BOOL;
   OP220_HomeONS : BOOL;
   OP220_HomingSeq : udt_SequenceStructure_X64 := (CycleDone := 1, CurrentStep := 9000, NextStep := 9000, ONS := -32768, StepHistory[0] := 1140, StepHistory[1] := 9000, StepHistory[2] := 1000, StepHistory[3] := 1020, StepHistory[4] := 1030, StepHistory[5] := 1140, StepHistory[6] := 9000, StepHistory[7] := 1000, StepHistory[8] := 1020, StepHistory[9] := 1030, StepHistory[10] := 1120, StepHistory[11] := 1140, StepHistory[12] := 9000, StepHistory[13] := 1000, StepHistory[14] := 1010, StepHistory[15] := 1020, StepHistory[16] := 1030, StepHistory[17] := 1120, StepHistory[18] := 1140, StepHistory[19] := 9000, StepHistory[20] := 1000, StepHistory[21] := 1020, StepHistory[22] := 1030, StepHistory[23] := 1120, StepHistory[24] := 1140, StepHistory[25] := 9000, StepHistory[26] := 1000, StepHistory[27] := 1020, StepHistory[28] := 1030, StepHistory[29] := 1140, StepHistory[30] := 1160, StepHistory[31] := 9000, StepHistory[32] := 1000, StepHistory[33] := 1020, StepHistory[34] := 1030, StepHistory[35] := 1140, StepHistory[36] := 1160, StepHistory[37] := 9000, StepHistory[38] := 1000, StepHistory[39] := 1020, StepHistory[40] := 1030, StepHistory[41] := 1140, StepHistory[42] := 1160, StepHistory[43] := 9000, StepHistory[44] := 1000, StepHistory[45] := 1020, StepHistory[46] := 1030, StepHistory[47] := 1120, StepHistory[48] := 1140, StepHistory[49] := 1160, StepHistory[50] := 9000, StepHistory[51] := 1000, StepHistory[52] := 1020, StepHistory[53] := 1030, StepHistory[54] := 1120, StepHistory[55] := 1140,
        StepHistory[56] := 1160, StepHistory[57] := 9000, StepHistory[58] := 1000, StepHistory[59] := 1020, StepHistory[60] := 1030, StepHistory[61] := 1120, StepHistory[62] := 1140, StepHistory[63] := 1160, StepDescriptionPointer := 1, CurrentCycleTime := 0.032, AverageCycleTime := 0.023, CycleTimeHistory[0] := 0.041, CycleTimeHistory[1] := 0.005, CycleTimeHistory[2] := 0.004, CycleTimeHistory[3] := 0.057, CycleTimeHistory[5] := 0.048, CycleTimeHistory[7] := 0.043, CycleTimeHistory[9] := 0.032, CurrentStepCycleTime := 0.028, StepTimeHistory[0] := 0.026, StepTimeHistory[1] := 0.026, StepTimeHistory[2] := 0.026, StepTimeHistory[3] := 0.026, StepTimeHistory[4] := 0.026, StepTimeHistory[5] := 0.026, StepTimeHistory[6] := 0.026, StepTimeHistory[7] := 0.026, StepTimeHistory[8] := 0.026, StepTimeHistory[9] := 0.026, StepTimeHistory[10] := 0.056, StepTimeHistory[11] := 0.056, StepTimeHistory[12] := 0.056, StepTimeHistory[13] := 0.037, StepTimeHistory[14] := 2.088, StepTimeHistory[15] := 2.088, StepTimeHistory[16] := 2.088, StepTimeHistory[17] := 0.037, StepTimeHistory[18] := 0.037, StepTimeHistory[23] := 0.038, StepTimeHistory[24] := 0.038, StepTimeHistory[25] := 0.038, StepTimeHistory[26] := 0.038, StepTimeHistory[27] := 0.038, StepTimeHistory[28] := 0.038, StepTimeHistory[29] := 0.038, StepTimeHistory[30] := 0.038, StepTimeHistory[31] := 0.038, StepTimeHistory[32] := 0.038, StepTimeHistory[33] := 0.038, StepTimeHistory[34] := 0.038, StepTimeHistory[35] := 0.038, StepTimeHistory[36] := 0.038, StepTimeHistory[37] := 0.038, StepTimeHistory[38] := 0.038, StepTimeHistory[39] := 0.052, StepTimeHistory[40] := 0.052, StepTimeHistory[41] := 0.052, StepTimeHistory[42] := 0.052, StepTimeHistory[47] := 0.042, StepTimeHistory[48] := 0.042,
        StepTimeHistory[49] := 0.042, StepTimeHistory[54] := 0.038, StepTimeHistory[55] := 0.038, StepTimeHistory[56] := 0.038, StepTimeHistory[61] := 0.028, StepTimeHistory[62] := 0.028, StepTimeHistory[63] := 0.028, StepTimer.PRE := 999999999, CycleTimer.PRE := 999999999);
   OP220_LeakTest : udt_ProcessFault;
   OP220_PartToPartCycleTMR : TIMER := (PRE := 999999999);
   OP220_ProcessFaultsONS : DINT;
   OP220_Seq : udt_SequenceStructure_X64 := (CurrentStep := 2, ONS := 2, StepHistory[0] := 9000, StepHistory[1] := 1000, StepHistory[2] := 6050, StepHistory[3] := 9000, StepHistory[4] := 1000, StepHistory[5] := 6050, StepHistory[6] := 9000, StepHistory[7] := 1000, StepHistory[8] := 6050, StepHistory[9] := 9000, StepHistory[10] := 1000, StepHistory[11] := 6050, StepHistory[12] := 9000, StepHistory[13] := 1000, StepHistory[14] := 6050, StepHistory[15] := 9000, StepHistory[16] := 1000, StepHistory[17] := 6050, StepHistory[18] := 9000, StepHistory[19] := 1000, StepHistory[20] := 6050, StepHistory[21] := 9000, StepHistory[22] := 1000, StepHistory[23] := 6050, StepHistory[24] := 9000, StepHistory[25] := 1000, StepHistory[26] := 6050, StepHistory[27] := 9000, StepHistory[28] := 1000, StepHistory[29] := 6050, StepHistory[30] := 9000, StepHistory[31] := 1000, StepHistory[32] := 6050, StepHistory[33] := 9000, StepHistory[34] := 1000, StepHistory[35] := 6050, StepHistory[36] := 9000, StepHistory[37] := 1000, StepHistory[38] := 6050, StepHistory[39] := 9000, StepHistory[40] := 1000, StepHistory[41] := 6050, StepHistory[42] := 9000, StepHistory[43] := 1000, StepHistory[44] := 6050, StepHistory[45] := 9000, StepHistory[46] := 1000, StepHistory[47] := 6050, StepHistory[48] := 9000, StepHistory[49] := 1000, StepHistory[50] := 6050, StepHistory[51] := 9000, StepHistory[52] := 1000, StepHistory[53] := 6050, StepHistory[54] := 9000, StepHistory[55] := 1000, StepHistory[56] := 6050, StepHistory[57] := 9000,
        StepHistory[58] := 1000, StepHistory[59] := 6050, StepHistory[60] := 9000, StepHistory[61] := 1000, StepHistory[62] := 6050, StepHistory[63] := 9000, StepDescriptionPointer := 1, CurrentCycleTime := 0.001, AverageCycleTime := 0.0685, PreviousCycleTime := 0.002, CycleTimeHistory[0] := 0.002, CycleTimeHistory[1] := 0.002, CycleTimeHistory[2] := 0.001, CycleTimeHistory[3] := 0.001, CycleTimeHistory[4] := 0.001, CycleTimeHistory[5] := 0.002, CycleTimeHistory[6] := 0.002, CycleTimeHistory[7] := 0.671, CycleTimeHistory[8] := 0.002, CycleTimeHistory[9] := 0.001, CurrentStepCycleTime := 0.669, StepTimeHistory[0] := 0.217, StepTimeHistory[1] := 0.217, StepTimeHistory[2] := 0.217, StepTimeHistory[3] := 0.217, StepTimeHistory[4] := 0.217, StepTimeHistory[5] := 0.217, StepTimeHistory[6] := 0.217, StepTimeHistory[7] := 0.217, StepTimeHistory[8] := 0.217, StepTimeHistory[9] := 0.217, StepTimeHistory[10] := 0.217, StepTimeHistory[11] := 0.217, StepTimeHistory[12] := 0.217, StepTimeHistory[13] := 0.217, StepTimeHistory[14] := 0.217, StepTimeHistory[15] := 0.217, StepTimeHistory[16] := 0.217, StepTimeHistory[17] := 0.217, StepTimeHistory[18] := 0.217, StepTimeHistory[19] := 0.217, StepTimeHistory[20] := 0.217, StepTimeHistory[21] := 0.217, StepTimeHistory[22] := 0.217, StepTimeHistory[23] := 0.217, StepTimeHistory[24] := 0.217, StepTimeHistory[25] := 0.217, StepTimeHistory[26] := 0.217, StepTimeHistory[27] := 0.217, StepTimeHistory[28] := 0.217, StepTimeHistory[29] := 0.217, StepTimeHistory[30] := 0.217, StepTimeHistory[31] := 0.217, StepTimeHistory[32] := 0.217, StepTimeHistory[33] := 0.217, StepTimeHistory[34] := 0.217, StepTimeHistory[35] := 0.217, StepTimeHistory[36] := 0.217, StepTimeHistory[37] := 0.217, StepTimeHistory[38] := 0.217,
        StepTimeHistory[39] := 0.217, StepTimeHistory[40] := 0.217, StepTimeHistory[41] := 0.217, StepTimeHistory[42] := 0.217, StepTimeHistory[43] := 0.217, StepTimeHistory[44] := 0.217, StepTimeHistory[45] := 0.217, StepTimeHistory[46] := 0.217, StepTimeHistory[47] := 0.217, StepTimeHistory[48] := 0.217, StepTimeHistory[49] := 0.217, StepTimeHistory[50] := 0.217, StepTimeHistory[51] := 0.217, StepTimeHistory[52] := 0.217, StepTimeHistory[53] := 0.217, StepTimeHistory[54] := 0.217, StepTimeHistory[55] := 0.669, StepTimeHistory[56] := 0.669, StepTimeHistory[57] := 0.669, StepTimeHistory[58] := 0.669, StepTimeHistory[59] := 0.669, StepTimeHistory[60] := 0.669, StepTimeHistory[61] := 0.669, StepTimeHistory[62] := 0.669, StepTimeHistory[63] := 0.669, StepTimer.PRE := 999999999, CycleTimer.PRE := 999999999);
   OutfeedCounter : COUNTER := (PRE := 9999999, ACC := 26195);
   ResetFeedCounters : BOOL;
   RFID_Comp : AOI_RFIDCompare;
   RFID_DiagData : DINT[4];
   RFID_EntryStatus : DINT;
   RFID_ExpectedFixtureVal : SINT[5,12] := ([1,0] := 26, [1,1] := 6, [1,2] := 2, [1,3] := 26, [1,5] := 7, [1,6] := 4, [1,7] := 1, [1,8] := 3, [1,10] := 1, [1,11] := 1, [2,0] := 26, [2,1] := 6, [2,2] := 2, [2,3] := 26, [2,5] := 7, [2,6] := 4, [2,7] := 1, [2,8] := 4, [2,10] := 2, [2,11] := 2);
   RFID_FaultCode : DINT;
   RFID_ReceiveBuffer : SINT[8000];
   RFID_RWHPort1 : RWH_CMD := (isiModuleID := 13, isiFunctionID := 4, iiRdWrLength := 40);
   RFID_RWHPort2 : RWH_CMD := (isiModuleID := 13, iiInputStartAdd := 46, iiOutputStartAdd := 46, isiFunctionID := 4, iiRdWrLength := 40);
   RFID_SendBuffer : SINT[8000];
   RFIDScanner : udt_OutputStructure := (REQ := 1);
   RFIDTag1Match : BOOL;
   RFIDTag2Match : BOOL;
   Robot : udt_OutputStructure := (IL := 1, BC := 1, REQ := 1);
   RobotGripper : udt_OutputStructure := (IL := 1, BTMR.PRE := 2000);
   RobotInputs : udt_EpsonInputs := (ib_Ready := 1, ib_MotorsOn := 1, ib_InPos := 1, ib_GripOpen := 1, iB_SpeedEcho := 10, iW_PositionEcho := 1, iR_X := 149.65157, iR_Y := 115.6004, iR_Z := -29.66788, iR_U := 57.989914);
   RobotOutputs : udt_EpsonOutputs := (ob_SpeedOverride := 1, oB_SpeedPerc := 10, oW_TargetPosition := 1, oR_X := 191.0, oR_Y := -84.0, oR_Z := -52.0, oR_U := -270.0);
   ShiftTimes : SINT[24] := ([0] := 7, [1] := 15, [2] := 23, [3] := -1, [4] := -1, [5] := -1, [6] := -1, [7] := -1, [8] := -1, [9] := -1, [10] := -1, [11] := -1, [12] := -1, [13] := -1, [14] := -1, [15] := -1, [16] := -1, [17] := -1, [18] := -1, [19] := -1, [20] := -1, [21] := -1, [22] := -1, [23] := -1);
   TempConsumedFromPLC : BOOL;
   TempStrBuff : STRING[10] := ([0] := '9000', [1] := '/', [2] := '0', [3] := ')');
   test : BOOL;
   TON_CapActuatorsDelay : TIMER := (PRE := 5000);
   TON_CapActuatorsDelay2 : TIMER := (PRE := 100);
   TON_CapCTSDelay : TIMER := (PRE := 2000);
   TON_CapCTSDelay2 : TIMER := (PRE := 2000);
   TON_CapCylindersDelay : TIMER := (PRE := 5500);
   TON_CapShuffleCTS1Delay : TIMER := (PRE := 5000);
   TON_CapShuffleCTS2Delay : TIMER := (PRE := 5000);
   TON_ConveyorCleatTimeout : TIMER := (PRE := 5000);
   TON_ConvUnloadDelay : TIMER := (PRE := 300, ACC := 300, EN := 1, DN := 1);
   TON_CTS1GetResultRetry : TIMER := (PRE := 1000);
   TON_CTS1GetResultTimeout : TIMER := (PRE := 1000);
   TON_CTS1NotGettingResultsTimeout : TIMER := (PRE := 1000);
   TON_CTS1Trigger0 : TIMER := (PRE := 200);
   TON_CTS1Trigger1 : TIMER := (PRE := 200);
   TON_CTS1Trigger2 : TIMER := (PRE := 200);
   TON_CTS2GetResultRetry : TIMER := (PRE := 1000);
   TON_CTS2GetResultTimeout : TIMER := (PRE := 1000);
   TON_CTS2NotGettingResultsTimeout : TIMER := (PRE := 1000);
   TON_CTS2Trigger0 : TIMER := (PRE := 200);
   TON_CTS2Trigger1 : TIMER := (PRE := 200);
   TON_CTS2Trigger2 : TIMER := (PRE := 1000);
   TON_Cylinder1DownTimeout : TIMER := (PRE := 5000);
   TON_Cylinder1UpTimeout : TIMER := (PRE := 5000);
   TON_Cylinder2DownTimeout : TIMER := (PRE := 5000);
   TON_Cylinder2UpTimeout : TIMER := (PRE := 5000);
   TON_FailChute : TIMER[10] := ([0].PRE := 1000, [1].PRE := 1000, [2].PRE := 1000, [3].PRE := 1000);
   TON_HMICloseDisplayDelay : TIMER := (PRE := 500);
   TON_Nest1CylinderTimer : TIMER := (PRE := 5000);
   TON_Nest1DryCycleDryTest : TIMER := (PRE := 5000);
   TON_Nest2CylinderTimer : TIMER := (PRE := 5000);
   TON_Nest2DryCycleDryTest : TIMER := (PRE := 5000);
   TON_RobotPickupSafeDelay : TIMER := (PRE := 200, ACC := 500, EN := 1, DN := 1);
   TON_RobotReqRetry : TIMER := (PRE := 1000);
   TON_RobotReqTimeout : TIMER := (PRE := 1000);
END_VAR

ROUTINE AManualDebug   (* ladder *)
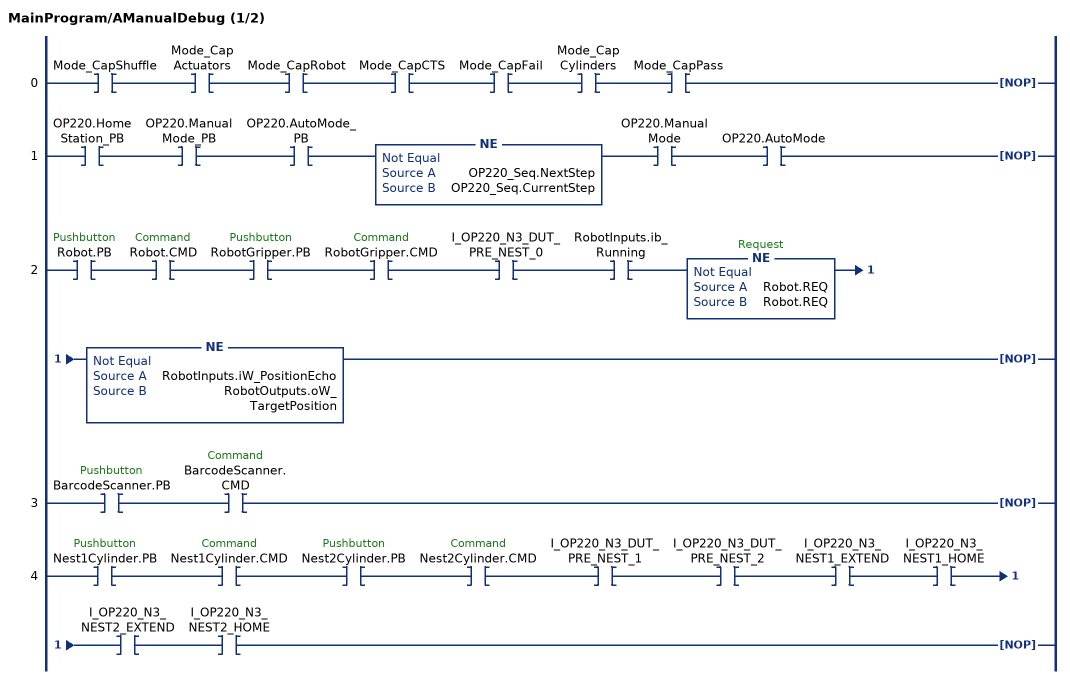
   [picture p27: MainProgram/AManualDebug rungs 0-4]
   0: XIC(Mode_CapShuffle)XIC(Mode_CapActuators)XIC(Mode_CapRobot)XIC(Mode_CapCTS)XIC(Mode_CapFail)XIC(Mode_CapCylinders)XIC(Mode_CapPass)NOP();
   1: XIC(OP220.HomeStation_PB)XIC(OP220.ManualMode_PB)XIC(OP220.AutoMode_PB)NE(OP220_Seq.NextStep,OP220_Seq.CurrentStep)XIC(OP220.ManualMode)XIC(OP220.AutoMode)NOP();
   2: XIC(Robot.PB)XIC(Robot.CMD)XIC(RobotGripper.PB)XIC(RobotGripper.CMD)XIC(I_OP220_N3_DUT_PRE_NEST_0)XIC(RobotInputs.ib_Running)NE(Robot.REQ,Robot.REQ)NE(RobotInputs.iW_PositionEcho,RobotOutputs.oW_TargetPosition)NOP();
   3: XIC(BarcodeScanner.PB)XIC(BarcodeScanner.CMD)NOP();
   4: XIC(Nest1Cylinder.PB)XIC(Nest1Cylinder.CMD)XIC(Nest2Cylinder.PB)XIC(Nest2Cylinder.CMD)XIC(I_OP220_N3_DUT_PRE_NEST_1)XIC(I_OP220_N3_DUT_PRE_NEST_2)XIC(I_OP220_N3_NEST1_EXTEND)XIC(I_OP220_N3_NEST1_HOME)XIC(I_OP220_N3_NEST2_EXTEND)XIC(I_OP220_N3_NEST2_HOME)NOP();
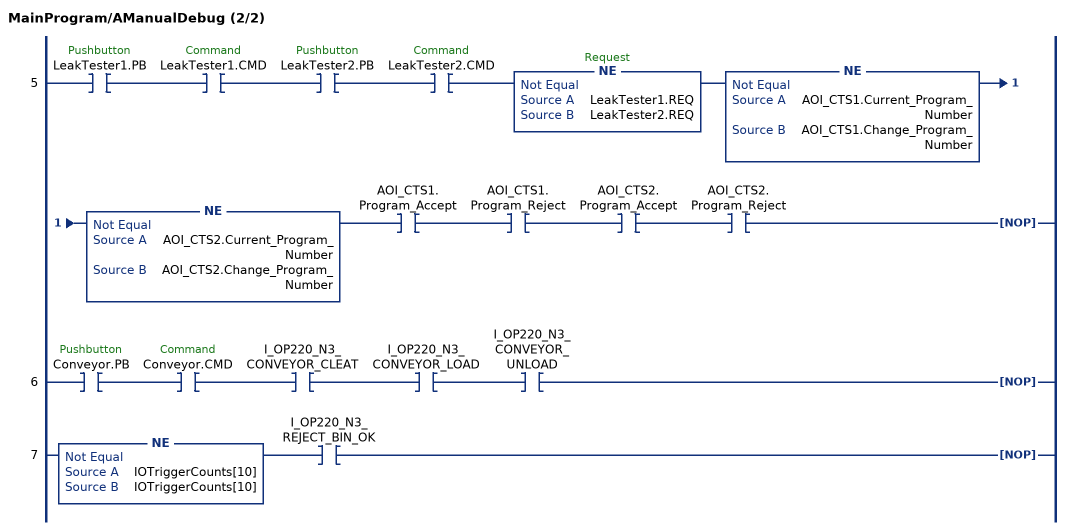
   5: XIC(LeakTester1.PB)XIC(LeakTester1.CMD)XIC(LeakTester2.PB)XIC(LeakTester2.CMD)NE(LeakTester1.REQ,LeakTester2.REQ)NE(AOI_CTS1.Current_Program_Number,AOI_CTS1.Change_Program_Number)NE(AOI_CTS2.Current_Program_Number,AOI_CTS2.Change_Program_Number)XIC(AOI_CTS1.Program_Accept)XIC(AOI_CTS1.Program_Reject)XIC(AOI_CTS2.Program_Accept)XIC(AOI_CTS2.Program_Reject)NOP();
   6: XIC(Conveyor.PB)XIC(Conveyor.CMD)XIC(I_OP220_N3_CONVEYOR_CLEAT)XIC(I_OP220_N3_CONVEYOR_LOAD)XIC(I_OP220_N3_CONVEYOR_UNLOAD)NOP();
   7: NE(IOTriggerCounts[10],IOTriggerCounts[10])XIC(I_OP220_N3_REJECT_BIN_OK)NOP();
END_ROUTINE

ROUTINE MainRoutine   (* ladder *)
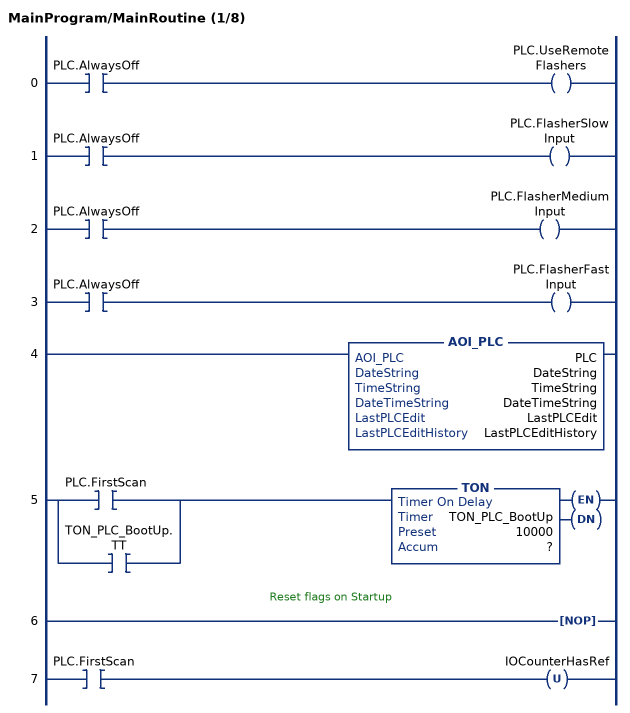
   0: XIC(PLC.AlwaysOff)OTE(PLC.UseRemoteFlashers);
   1: XIC(PLC.AlwaysOff)OTE(PLC.FlasherSlowInput);
   2: XIC(PLC.AlwaysOff)OTE(PLC.FlasherMediumInput);
   3: XIC(PLC.AlwaysOff)OTE(PLC.FlasherFastInput);
   4: AOI_PLC(PLC,DateString,TimeString,DateTimeString,LastPLCEdit,LastPLCEditHistory);
   5: [XIC(PLC.FirstScan) ,XIC(TON_PLC_BootUp.TT) ]TON(TON_PLC_BootUp,?,?);
   // Reset flags on Startup
   6: NOP();
   7: XIC(PLC.FirstScan)OTU(IOCounterHasRef);
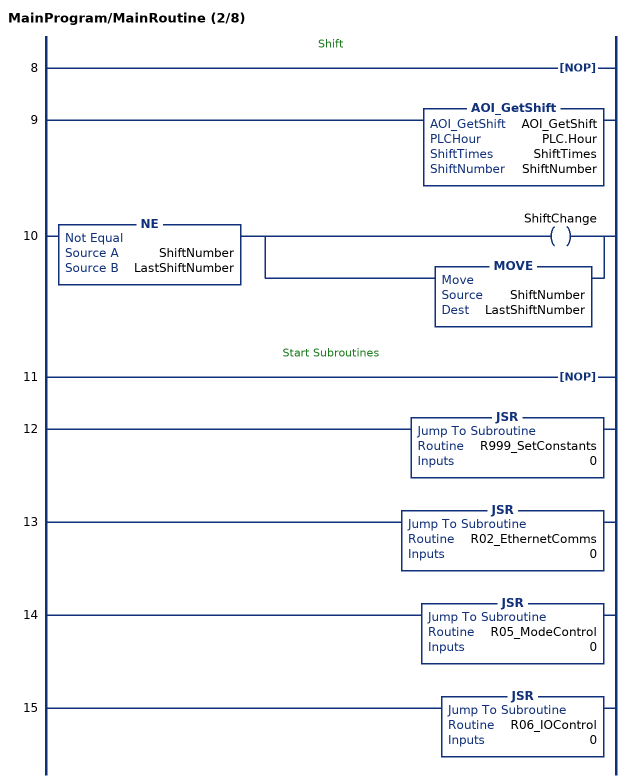
   // Shift
   8: NOP();
   9: AOI_GetShift(AOI_GetShift,PLC.Hour,ShiftTimes,ShiftNumber);
   10: NE(ShiftNumber,LastShiftNumber)[OTE(ShiftChange) ,MOVE(ShiftNumber,LastShiftNumber) ];
   // Start Subroutines
   11: NOP();
   12: JSR(R999_SetConstants,0);
   13: JSR(R02_EthernetComms,0);
   14: JSR(R05_ModeControl,0);
   15: JSR(R06_IOControl,0);
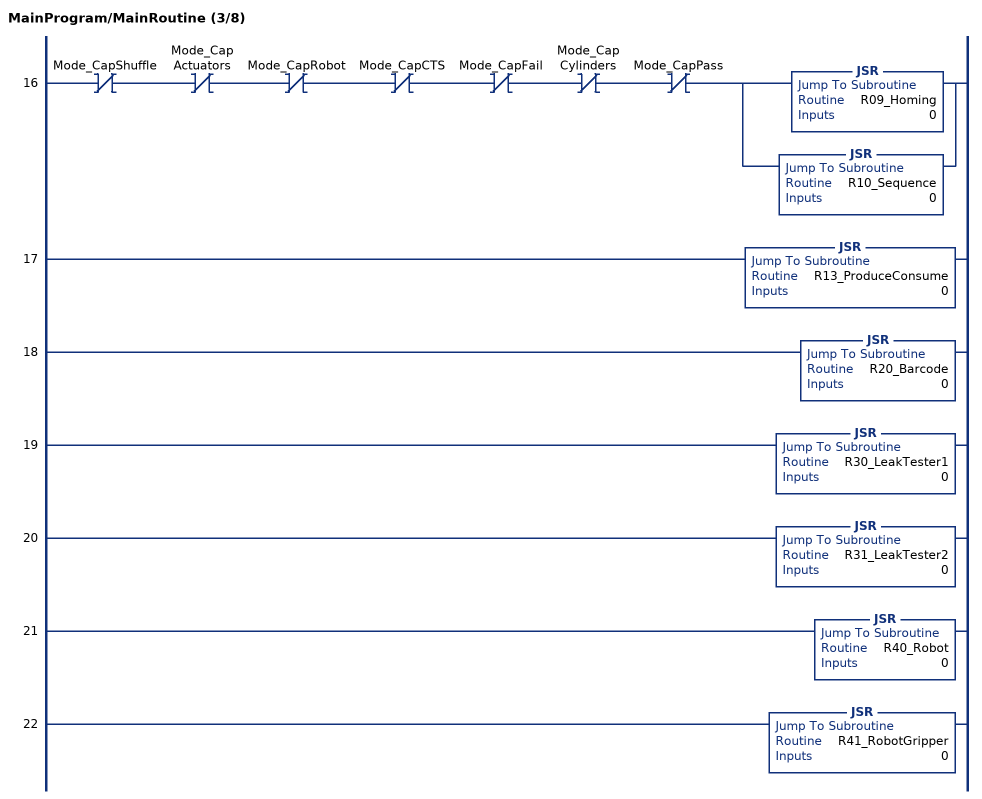
   16: XIO(Mode_CapShuffle)XIO(Mode_CapActuators)XIO(Mode_CapRobot)XIO(Mode_CapCTS)XIO(Mode_CapFail)XIO(Mode_CapCylinders)XIO(Mode_CapPass)[JSR(R09_Homing,0) ,JSR(R10_Sequence,0) ];
   17: JSR(R13_ProduceConsume,0);
   18: JSR(R20_Barcode,0);
   19: JSR(R30_LeakTester1,0);
   20: JSR(R31_LeakTester2,0);
   21: JSR(R40_Robot,0);
   22: JSR(R41_RobotGripper,0);
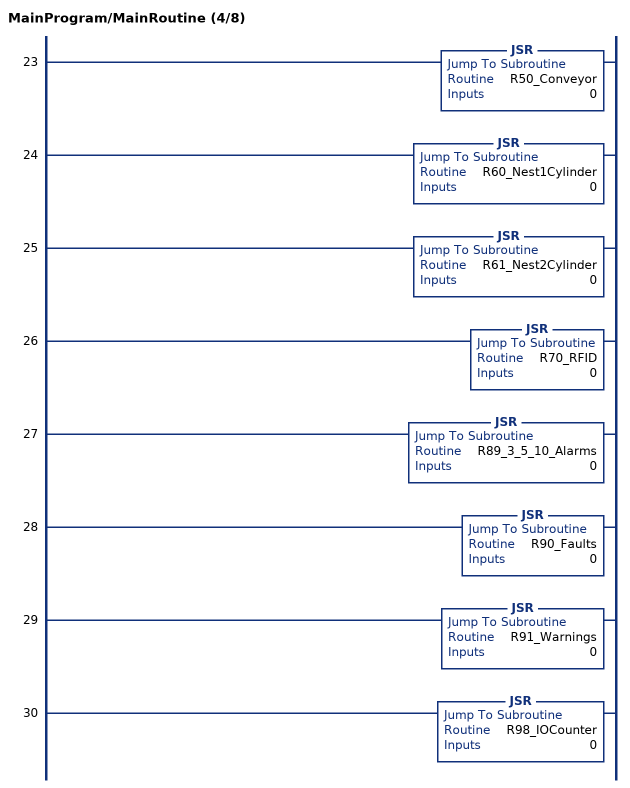
   23: JSR(R50_Conveyor,0);
   24: JSR(R60_Nest1Cylinder,0);
   25: JSR(R61_Nest2Cylinder,0);
   26: JSR(R70_RFID,0);
   27: JSR(R89_3_5_10_Alarms,0);
   28: JSR(R90_Faults,0);
   29: JSR(R91_Warnings,0);
   30: JSR(R98_IOCounter,0);
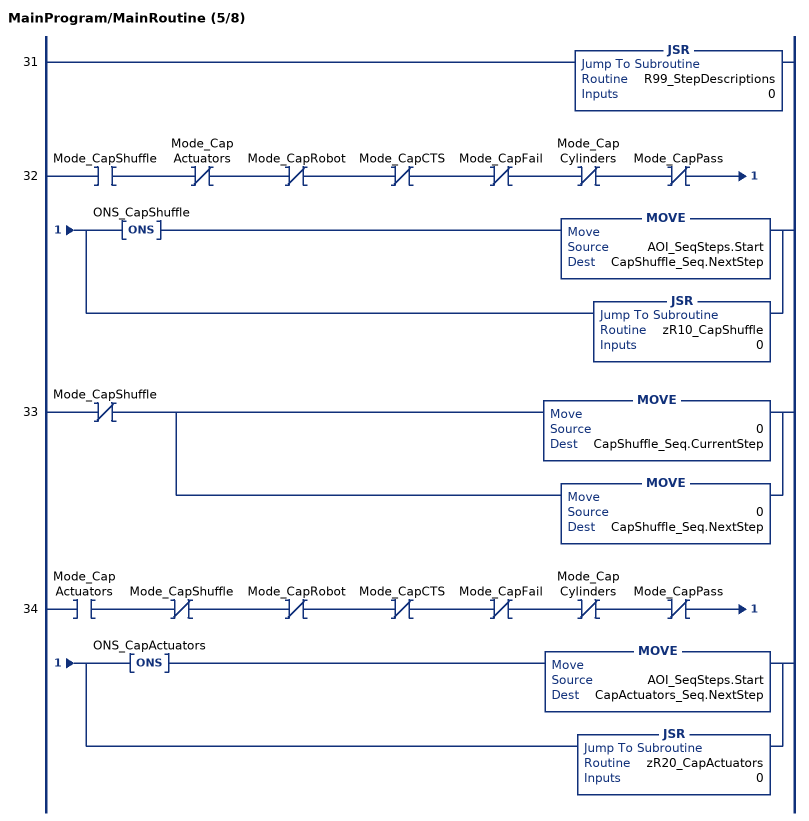
   31: JSR(R99_StepDescriptions,0);
   32: XIC(Mode_CapShuffle)XIO(Mode_CapActuators)XIO(Mode_CapRobot)XIO(Mode_CapCTS)XIO(Mode_CapFail)XIO(Mode_CapCylinders)XIO(Mode_CapPass)[ONS(ONS_CapShuffle) MOVE(AOI_SeqSteps.Start,CapShuffle_Seq.NextStep) ,JSR(zR10_CapShuffle,0) ];
   33: XIO(Mode_CapShuffle)[MOVE(0,CapShuffle_Seq.CurrentStep) ,MOVE(0,CapShuffle_Seq.NextStep) ];
   34: XIC(Mode_CapActuators)XIO(Mode_CapShuffle)XIO(Mode_CapRobot)XIO(Mode_CapCTS)XIO(Mode_CapFail)XIO(Mode_CapCylinders)XIO(Mode_CapPass)[ONS(ONS_CapActuators) MOVE(AOI_SeqSteps.Start,CapActuators_Seq.NextStep) ,JSR(zR20_CapActuators,0) ];
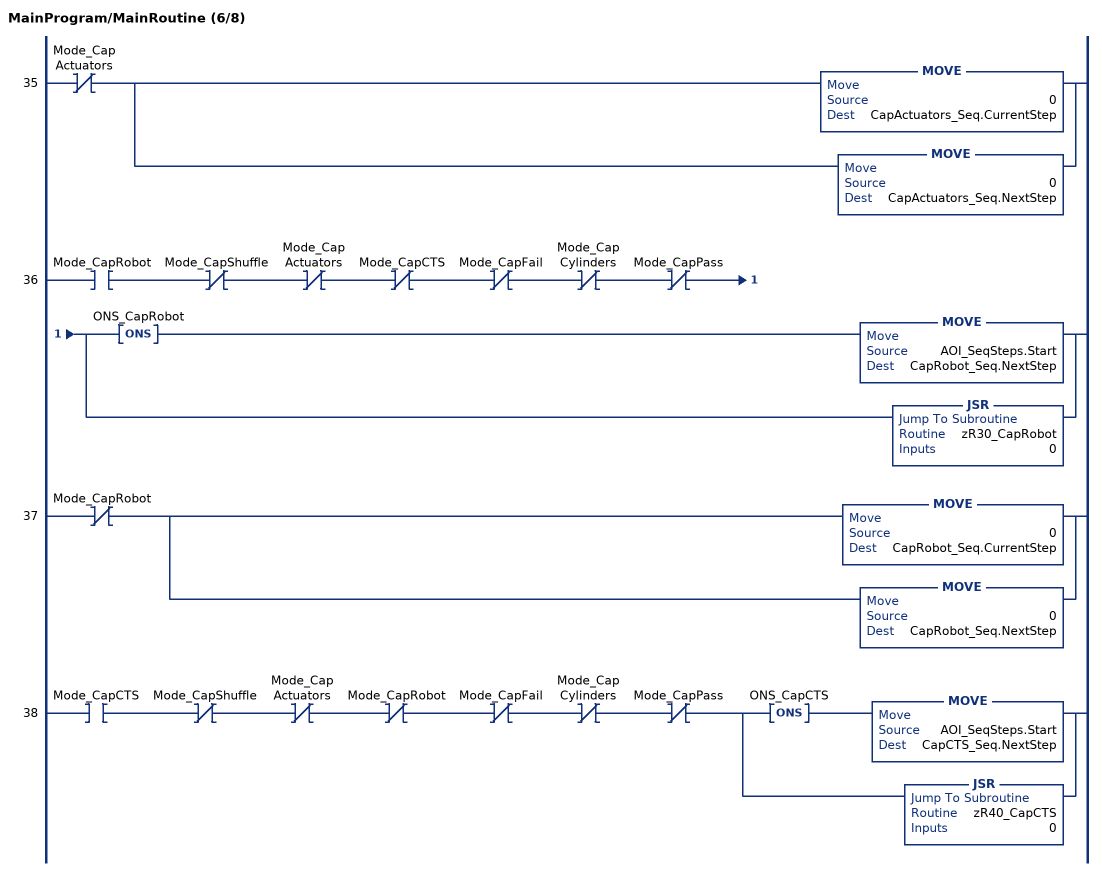
   35: XIO(Mode_CapActuators)[MOVE(0,CapActuators_Seq.CurrentStep) ,MOVE(0,CapActuators_Seq.NextStep) ];
   36: XIC(Mode_CapRobot)XIO(Mode_CapShuffle)XIO(Mode_CapActuators)XIO(Mode_CapCTS)XIO(Mode_CapFail)XIO(Mode_CapCylinders)XIO(Mode_CapPass)[ONS(ONS_CapRobot) MOVE(AOI_SeqSteps.Start,CapRobot_Seq.NextStep) ,JSR(zR30_CapRobot,0) ];
   37: XIO(Mode_CapRobot)[MOVE(0,CapRobot_Seq.CurrentStep) ,MOVE(0,CapRobot_Seq.NextStep) ];
   38: XIC(Mode_CapCTS)XIO(Mode_CapShuffle)XIO(Mode_CapActuators)XIO(Mode_CapRobot)XIO(Mode_CapFail)XIO(Mode_CapCylinders)XIO(Mode_CapPass)[ONS(ONS_CapCTS) MOVE(AOI_SeqSteps.Start,CapCTS_Seq.NextStep) ,JSR(zR40_CapCTS,0) ];
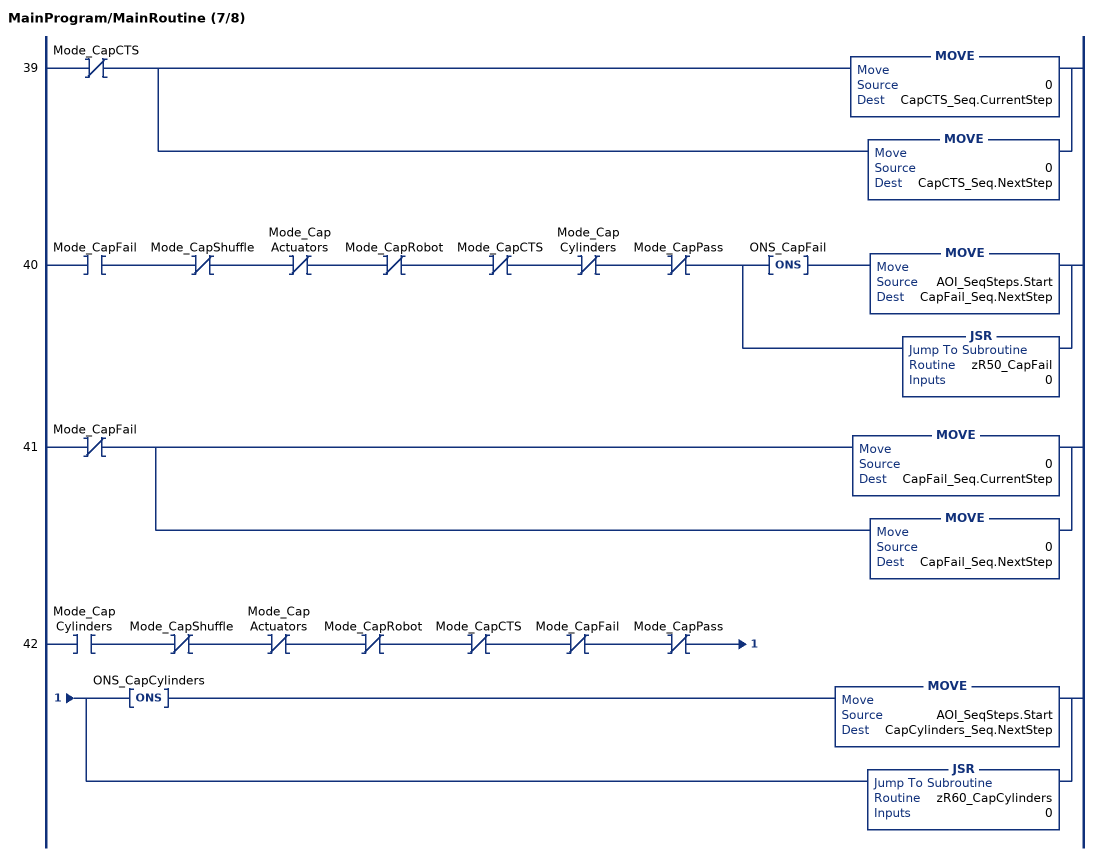
   39: XIO(Mode_CapCTS)[MOVE(0,CapCTS_Seq.CurrentStep) ,MOVE(0,CapCTS_Seq.NextStep) ];
   40: XIC(Mode_CapFail)XIO(Mode_CapShuffle)XIO(Mode_CapActuators)XIO(Mode_CapRobot)XIO(Mode_CapCTS)XIO(Mode_CapCylinders)XIO(Mode_CapPass)[ONS(ONS_CapFail) MOVE(AOI_SeqSteps.Start,CapFail_Seq.NextStep) ,JSR(zR50_CapFail,0) ];
   41: XIO(Mode_CapFail)[MOVE(0,CapFail_Seq.CurrentStep) ,MOVE(0,CapFail_Seq.NextStep) ];
   42: XIC(Mode_CapCylinders)XIO(Mode_CapShuffle)XIO(Mode_CapActuators)XIO(Mode_CapRobot)XIO(Mode_CapCTS)XIO(Mode_CapFail)XIO(Mode_CapPass)[ONS(ONS_CapCylinders) MOVE(AOI_SeqSteps.Start,CapCylinders_Seq.NextStep) ,JSR(zR60_CapCylinders,0) ];
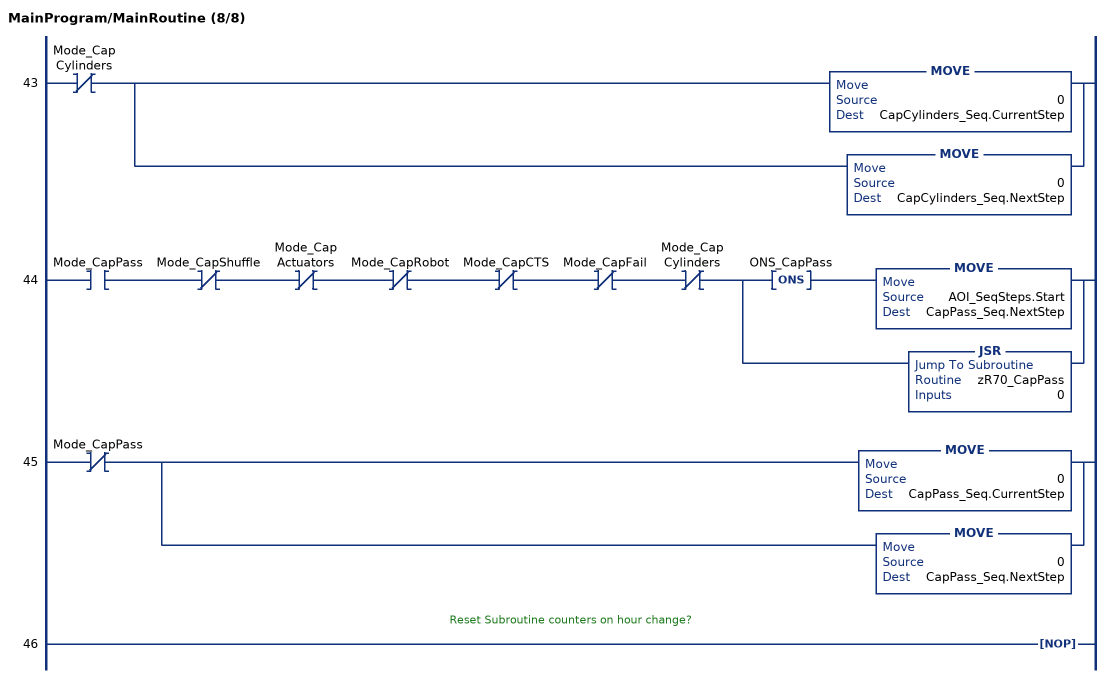
   43: XIO(Mode_CapCylinders)[MOVE(0,CapCylinders_Seq.CurrentStep) ,MOVE(0,CapCylinders_Seq.NextStep) ];
   44: XIC(Mode_CapPass)XIO(Mode_CapShuffle)XIO(Mode_CapActuators)XIO(Mode_CapRobot)XIO(Mode_CapCTS)XIO(Mode_CapFail)XIO(Mode_CapCylinders)[ONS(ONS_CapPass) MOVE(AOI_SeqSteps.Start,CapPass_Seq.NextStep) ,JSR(zR70_CapPass,0) ];
   45: XIO(Mode_CapPass)[MOVE(0,CapPass_Seq.CurrentStep) ,MOVE(0,CapPass_Seq.NextStep) ];
   // Reset Subroutine counters on hour change?
   46: NOP();
END_ROUTINE

ROUTINE R02_EthernetComms   (* ladder *)
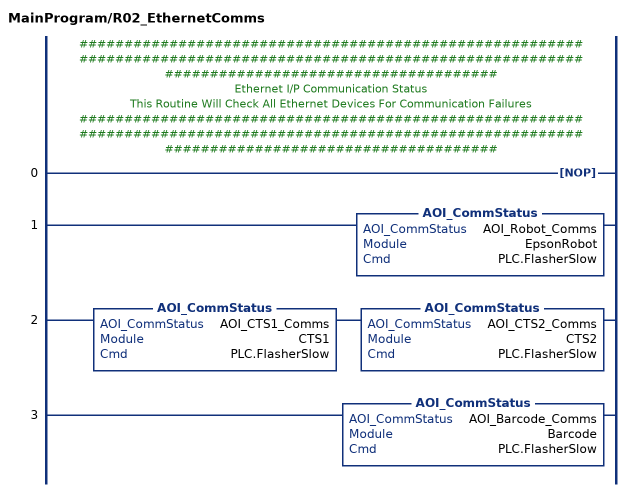
   // #####################################################################################################################################################
   // Ethernet I/P Communication Status
   // This Routine Will Check All Ethernet Devices For Communication Failures
   // #####################################################################################################################################################
   0: NOP();
   1: AOI_CommStatus(AOI_Robot_Comms,EpsonRobot,PLC.FlasherSlow);
   2: AOI_CommStatus(AOI_CTS1_Comms,CTS1,PLC.FlasherSlow)AOI_CommStatus(AOI_CTS2_Comms,CTS2,PLC.FlasherSlow);
   3: AOI_CommStatus(AOI_Barcode_Comms,Barcode,PLC.FlasherSlow);
END_ROUTINE

ROUTINE R05_ModeControl   (* ladder *)
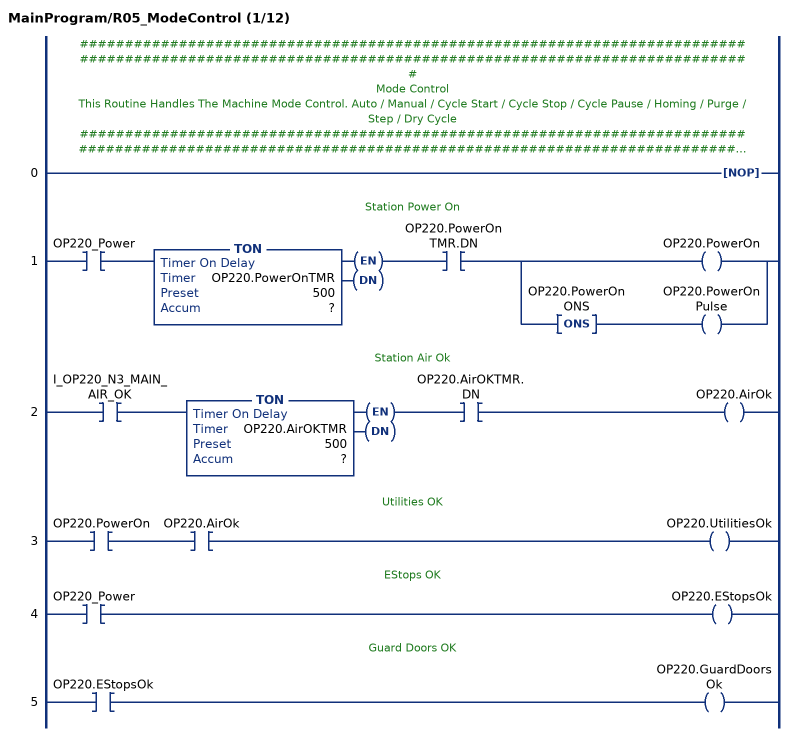
   // #####################################################################################################################################################
   // Mode Control
   // This Routine Handles The Machine Mode Control. Auto / Manual / Cycle Start / Cycle Stop / Cycle Pause / Homing / Purge / Step / Dry Cycle
   // #####################################################################################################################################################
   0: NOP();
   // Station Power On
   1: XIC(OP220_Power)TON(OP220.PowerOnTMR,?,?)XIC(OP220.PowerOnTMR.DN)[OTE(OP220.PowerOn) ,ONS(OP220.PowerOnONS) OTE(OP220.PowerOnPulse) ];
   // Station Air Ok
   2: XIC(I_OP220_N3_MAIN_AIR_OK)TON(OP220.AirOKTMR,?,?)XIC(OP220.AirOKTMR.DN)OTE(OP220.AirOk);
   // Utilities OK
   3: XIC(OP220.PowerOn)XIC(OP220.AirOk)OTE(OP220.UtilitiesOk);
   // EStops OK
   4: XIC(OP220_Power)OTE(OP220.EStopsOk);
   // Guard Doors OK
   5: XIC(OP220.EStopsOk)OTE(OP220.GuardDoorsOk);
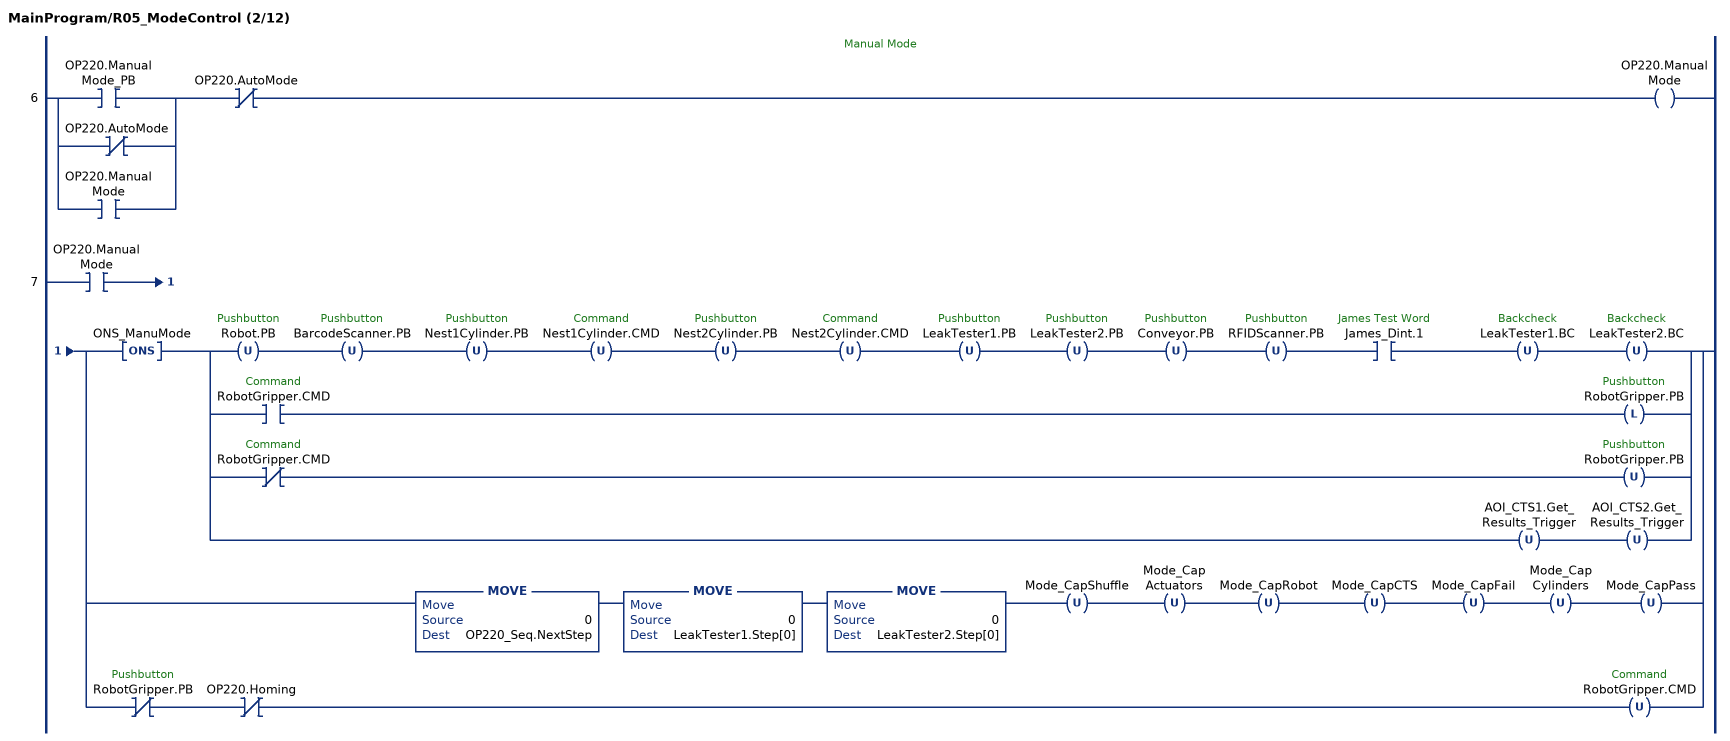
   // Manual Mode
   6: [XIC(OP220.ManualMode_PB) ,XIO(OP220.AutoMode) ,XIC(OP220.ManualMode) ]XIO(OP220.AutoMode)OTE(OP220.ManualMode);
   7: XIC(OP220.ManualMode)[ONS(ONS_ManuMode) [OTU(Robot.PB) OTU(BarcodeScanner.PB) OTU(Nest1Cylinder.PB) OTU(Nest1Cylinder.CMD) OTU(Nest2Cylinder.PB) OTU(Nest2Cylinder.CMD) OTU(LeakTester1.PB) OTU(LeakTester2.PB) OTU(Conveyor.PB) OTU(RFIDScanner.PB) XIC(James_Dint.1) OTU(LeakTester1.BC) OTU(LeakTester2.BC) ,XIC(RobotGripper.CMD) OTL(RobotGripper.PB) ,XIO(RobotGripper.CMD) OTU(RobotGripper.PB) ,OTU(AOI_CTS1.Get_Results_Trigger) OTU(AOI_CTS2.Get_Results_Trigger) ] ,MOVE(0,OP220_Seq.NextStep) MOVE(0,LeakTester1.Step[0]) MOVE(0,LeakTester2.Step[0]) OTU(Mode_CapShuffle) OTU(Mode_CapActuators) OTU(Mode_CapRobot) OTU(Mode_CapCTS) OTU(Mode_CapFail) OTU(Mode_CapCylinders) OTU(Mode_CapPass) ,XIO(RobotGripper.PB) XIO(OP220.Homing) OTU(RobotGripper.CMD) ];
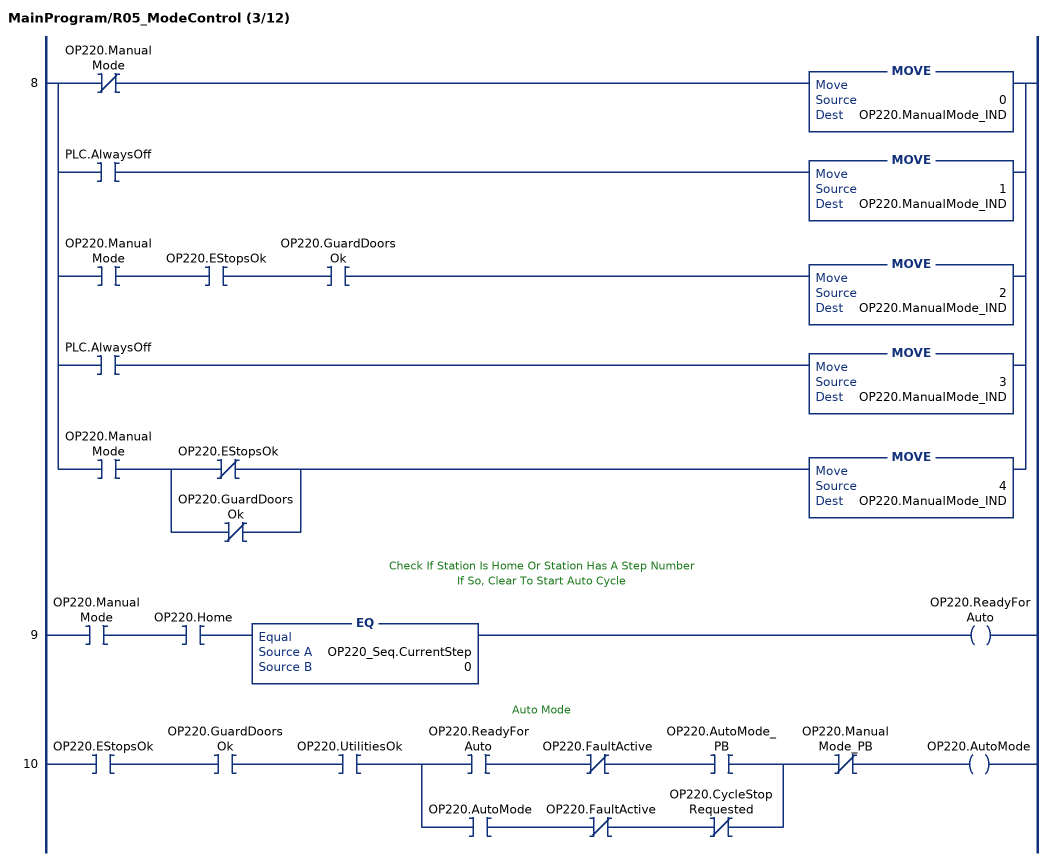
   8: [XIO(OP220.ManualMode) MOVE(0,OP220.ManualMode_IND) ,XIC(PLC.AlwaysOff) MOVE(1,OP220.ManualMode_IND) ,XIC(OP220.ManualMode) XIC(OP220.EStopsOk) XIC(OP220.GuardDoorsOk) MOVE(2,OP220.ManualMode_IND) ,XIC(PLC.AlwaysOff) MOVE(3,OP220.ManualMode_IND) ,XIC(OP220.ManualMode) [XIO(OP220.EStopsOk) ,XIO(OP220.GuardDoorsOk) ] MOVE(4,OP220.ManualMode_IND) ];
   // Check If Station Is Home Or Station Has A Step Number
   // If So, Clear To Start Auto Cycle
   9: XIC(OP220.ManualMode)XIC(OP220.Home)EQ(OP220_Seq.CurrentStep,0)OTE(OP220.ReadyForAuto);
   // Auto Mode
   10: XIC(OP220.EStopsOk)XIC(OP220.GuardDoorsOk)XIC(OP220.UtilitiesOk)[XIC(OP220.ReadyForAuto) XIO(OP220.FaultActive) XIC(OP220.AutoMode_PB) ,XIC(OP220.AutoMode) XIO(OP220.FaultActive) XIO(OP220.CycleStopRequested) ]XIO(OP220.ManualMode_PB)OTE(OP220.AutoMode);
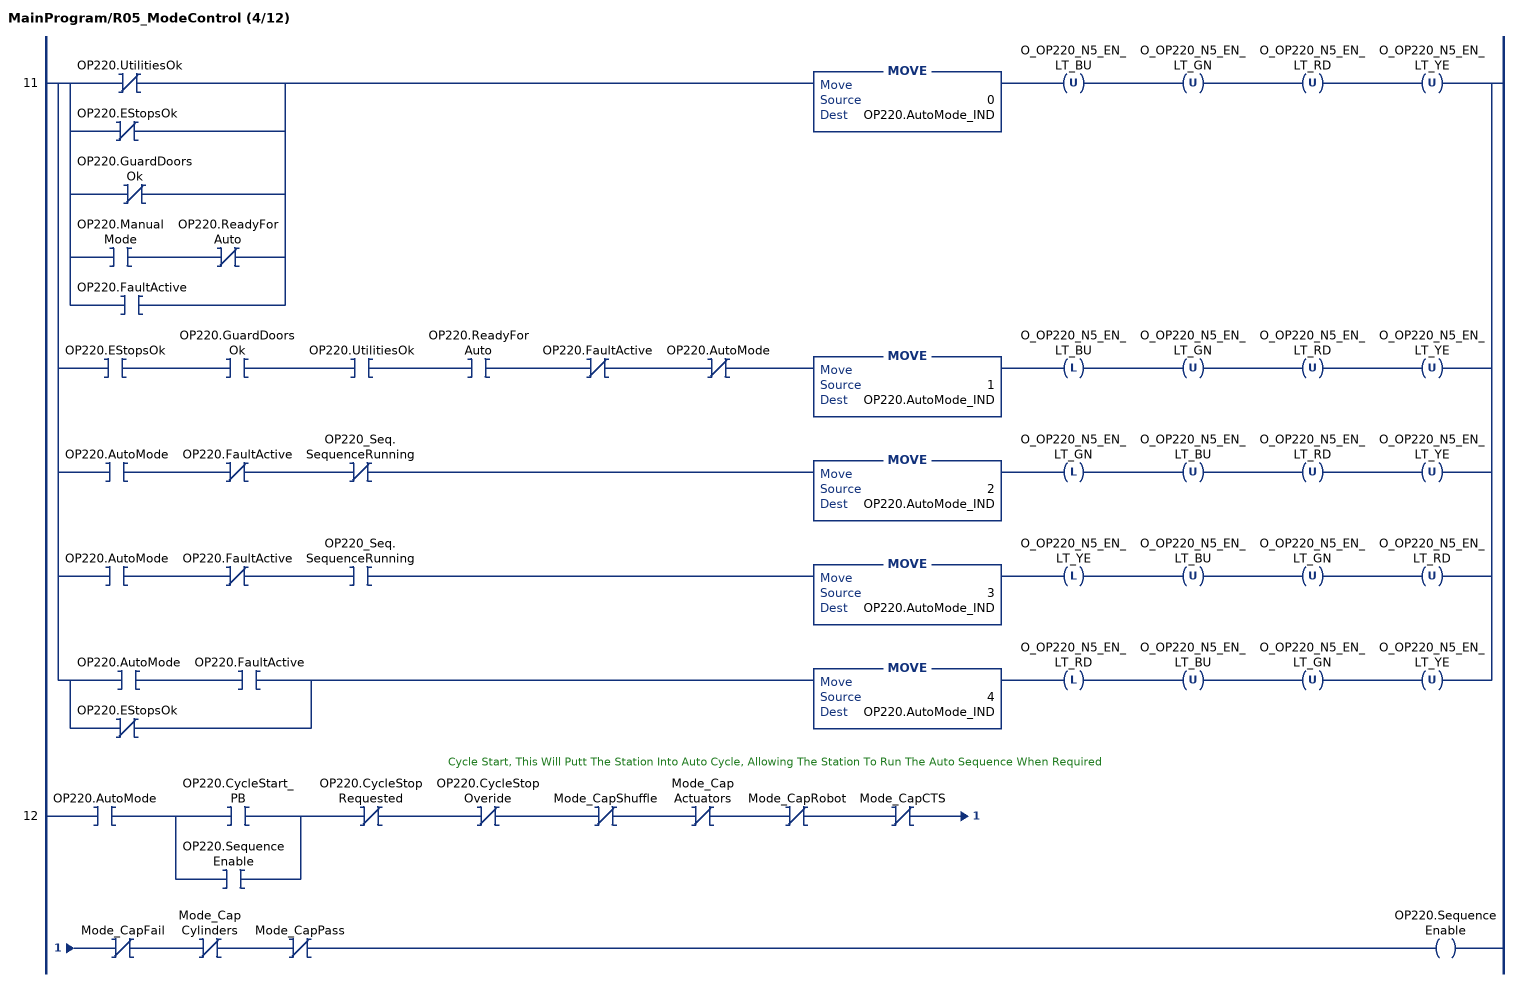
   11: [[XIO(OP220.UtilitiesOk) ,XIO(OP220.EStopsOk) ,XIO(OP220.GuardDoorsOk) ,XIC(OP220.ManualMode) XIO(OP220.ReadyForAuto) ,XIC(OP220.FaultActive) ] MOVE(0,OP220.AutoMode_IND) OTU(O_OP220_N5_EN_LT_BU) OTU(O_OP220_N5_EN_LT_GN) OTU(O_OP220_N5_EN_LT_RD) OTU(O_OP220_N5_EN_LT_YE) ,XIC(OP220.EStopsOk) XIC(OP220.GuardDoorsOk) XIC(OP220.UtilitiesOk) XIC(OP220.ReadyForAuto) XIO(OP220.FaultActive) XIO(OP220.AutoMode) MOVE(1,OP220.AutoMode_IND) OTL(O_OP220_N5_EN_LT_BU) OTU(O_OP220_N5_EN_LT_GN) OTU(O_OP220_N5_EN_LT_RD) OTU(O_OP220_N5_EN_LT_YE) ,XIC(OP220.AutoMode) XIO(OP220.FaultActive) XIO(OP220_Seq.SequenceRunning) MOVE(2,OP220.AutoMode_IND) OTL(O_OP220_N5_EN_LT_GN) OTU(O_OP220_N5_EN_LT_BU) OTU(O_OP220_N5_EN_LT_RD) OTU(O_OP220_N5_EN_LT_YE) ,XIC(OP220.AutoMode) XIO(OP220.FaultActive) XIC(OP220_Seq.SequenceRunning) MOVE(3,OP220.AutoMode_IND) OTL(O_OP220_N5_EN_LT_YE) OTU(O_OP220_N5_EN_LT_BU) OTU(O_OP220_N5_EN_LT_GN) OTU(O_OP220_N5_EN_LT_RD) ,[XIC(OP220.AutoMode) XIC(OP220.FaultActive) ,XIO(OP220.EStopsOk) ] MOVE(4,OP220.AutoMode_IND) OTL(O_OP220_N5_EN_LT_RD) OTU(O_OP220_N5_EN_LT_BU) OTU(O_OP220_N5_EN_LT_GN) OTU(O_OP220_N5_EN_LT_YE) ];
   // Cycle Start, This Will Putt The Station Into Auto Cycle, Allowing The Station To Run The Auto Sequence When Required
   12: XIC(OP220.AutoMode)[XIC(OP220.CycleStart_PB) ,XIC(OP220.SequenceEnable) ]XIO(OP220.CycleStopRequested)XIO(OP220.CycleStopOveride)XIO(Mode_CapShuffle)XIO(Mode_CapActuators)XIO(Mode_CapRobot)XIO(Mode_CapCTS)XIO(Mode_CapFail)XIO(Mode_CapCylinders)XIO(Mode_CapPass)OTE(OP220.SequenceEnable);
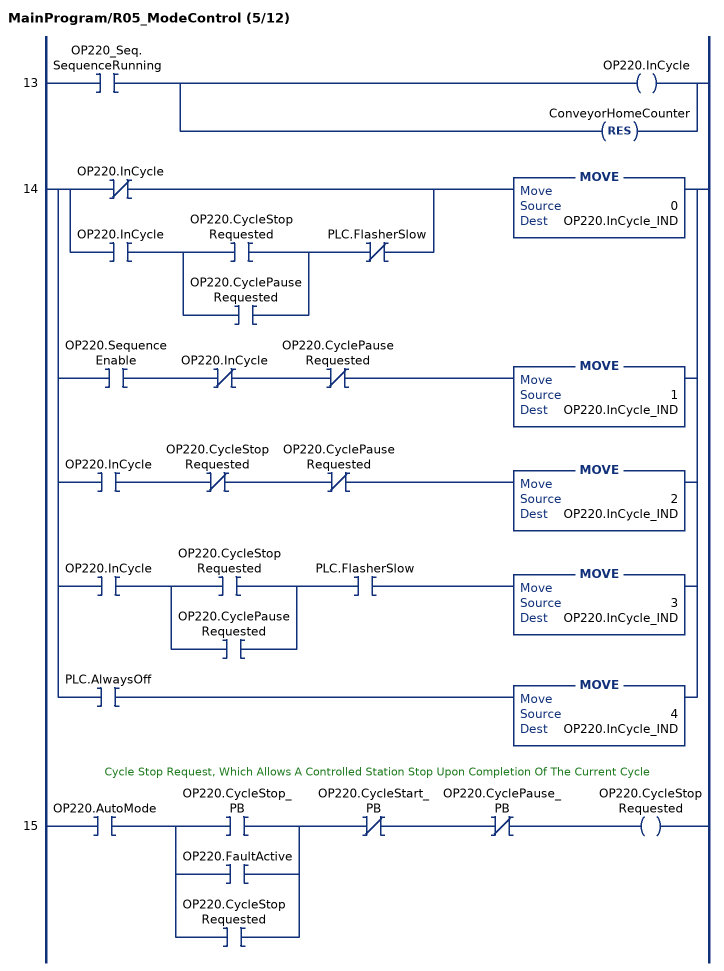
   13: XIC(OP220_Seq.SequenceRunning)[OTE(OP220.InCycle) ,RES(ConveyorHomeCounter) ];
   14: [[XIO(OP220.InCycle) ,XIC(OP220.InCycle) [XIC(OP220.CycleStopRequested) ,XIC(OP220.CyclePauseRequested) ] XIO(PLC.FlasherSlow) ] MOVE(0,OP220.InCycle_IND) ,XIC(OP220.SequenceEnable) XIO(OP220.InCycle) XIO(OP220.CyclePauseRequested) MOVE(1,OP220.InCycle_IND) ,XIC(OP220.InCycle) XIO(OP220.CycleStopRequested) XIO(OP220.CyclePauseRequested) MOVE(2,OP220.InCycle_IND) ,XIC(OP220.InCycle) [XIC(OP220.CycleStopRequested) ,XIC(OP220.CyclePauseRequested) ] XIC(PLC.FlasherSlow) MOVE(3,OP220.InCycle_IND) ,XIC(PLC.AlwaysOff) MOVE(4,OP220.InCycle_IND) ];
   // Cycle Stop Request, Which Allows A Controlled Station Stop Upon Completion Of The Current Cycle
   15: XIC(OP220.AutoMode)[XIC(OP220.CycleStop_PB) ,XIC(OP220.FaultActive) ,XIC(OP220.CycleStopRequested) ]XIO(OP220.CycleStart_PB)XIO(OP220.CyclePause_PB)OTE(OP220.CycleStopRequested);
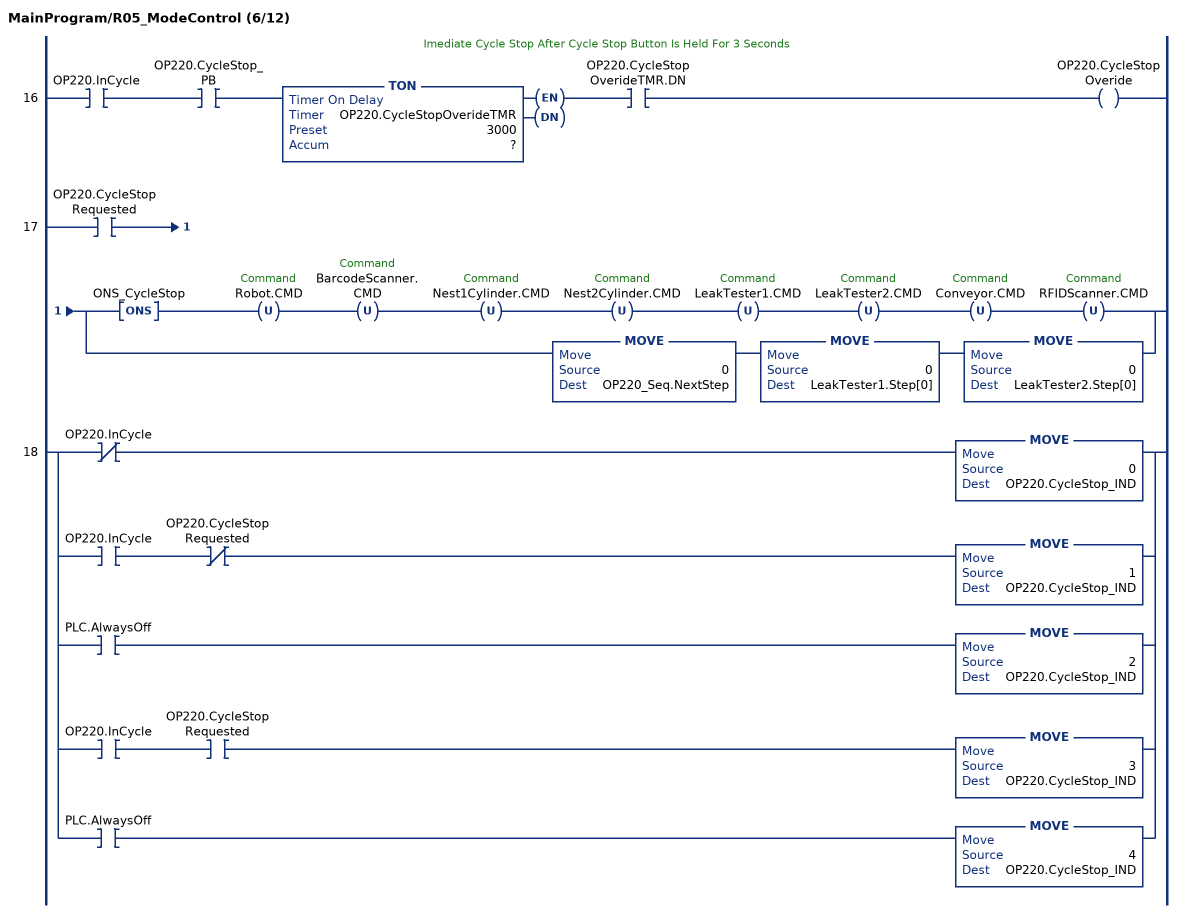
   // Imediate Cycle Stop After Cycle Stop Button Is Held For 3 Seconds
   16: XIC(OP220.InCycle)XIC(OP220.CycleStop_PB)TON(OP220.CycleStopOverideTMR,?,?)XIC(OP220.CycleStopOverideTMR.DN)OTE(OP220.CycleStopOveride);
   17: XIC(OP220.CycleStopRequested)[ONS(ONS_CycleStop) OTU(Robot.CMD) OTU(BarcodeScanner.CMD) OTU(Nest1Cylinder.CMD) OTU(Nest2Cylinder.CMD) OTU(LeakTester1.CMD) OTU(LeakTester2.CMD) OTU(Conveyor.CMD) OTU(RFIDScanner.CMD) ,MOVE(0,OP220_Seq.NextStep) MOVE(0,LeakTester1.Step[0]) MOVE(0,LeakTester2.Step[0]) ];
   18: [XIO(OP220.InCycle) MOVE(0,OP220.CycleStop_IND) ,XIC(OP220.InCycle) XIO(OP220.CycleStopRequested) MOVE(1,OP220.CycleStop_IND) ,XIC(PLC.AlwaysOff) MOVE(2,OP220.CycleStop_IND) ,XIC(OP220.InCycle) XIC(OP220.CycleStopRequested) MOVE(3,OP220.CycleStop_IND) ,XIC(PLC.AlwaysOff) MOVE(4,OP220.CycleStop_IND) ];
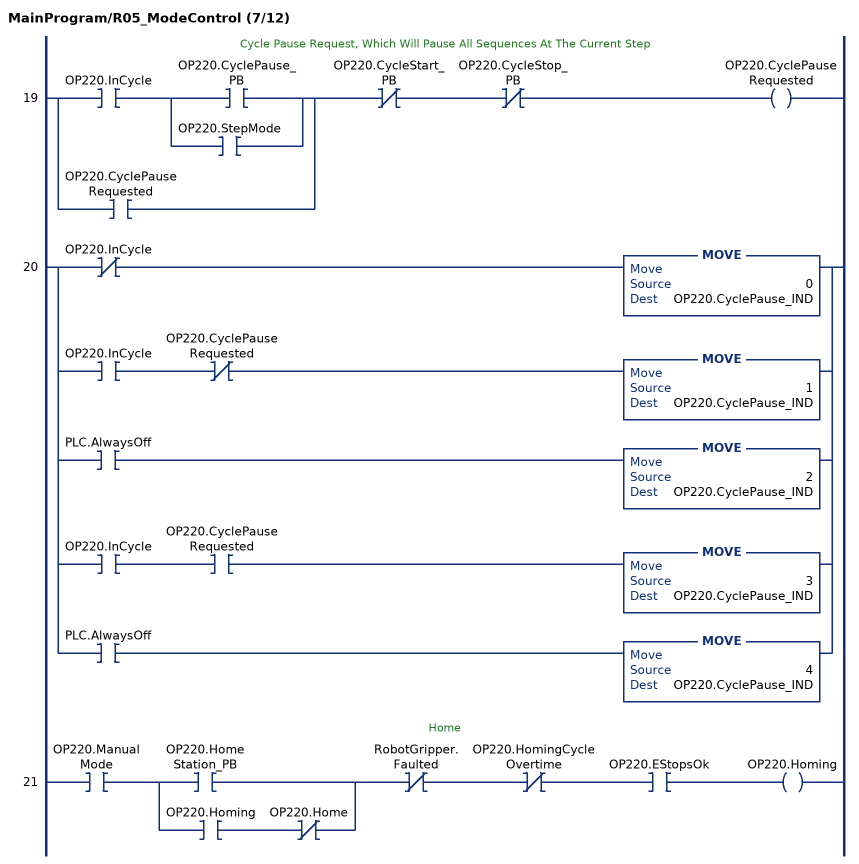
   // Cycle Pause Request, Which Will Pause All Sequences At The Current Step
   19: [XIC(OP220.InCycle) [XIC(OP220.CyclePause_PB) ,XIC(OP220.StepMode) ] ,XIC(OP220.CyclePauseRequested) ]XIO(OP220.CycleStart_PB)XIO(OP220.CycleStop_PB)OTE(OP220.CyclePauseRequested);
   20: [XIO(OP220.InCycle) MOVE(0,OP220.CyclePause_IND) ,XIC(OP220.InCycle) XIO(OP220.CyclePauseRequested) MOVE(1,OP220.CyclePause_IND) ,XIC(PLC.AlwaysOff) MOVE(2,OP220.CyclePause_IND) ,XIC(OP220.InCycle) XIC(OP220.CyclePauseRequested) MOVE(3,OP220.CyclePause_IND) ,XIC(PLC.AlwaysOff) MOVE(4,OP220.CyclePause_IND) ];
   // Home
   21: XIC(OP220.ManualMode)[XIC(OP220.HomeStation_PB) ,XIC(OP220.Homing) XIO(OP220.Home) ]XIO(RobotGripper.Faulted)XIO(OP220.HomingCycleOvertime)XIC(OP220.EStopsOk)OTE(OP220.Homing);
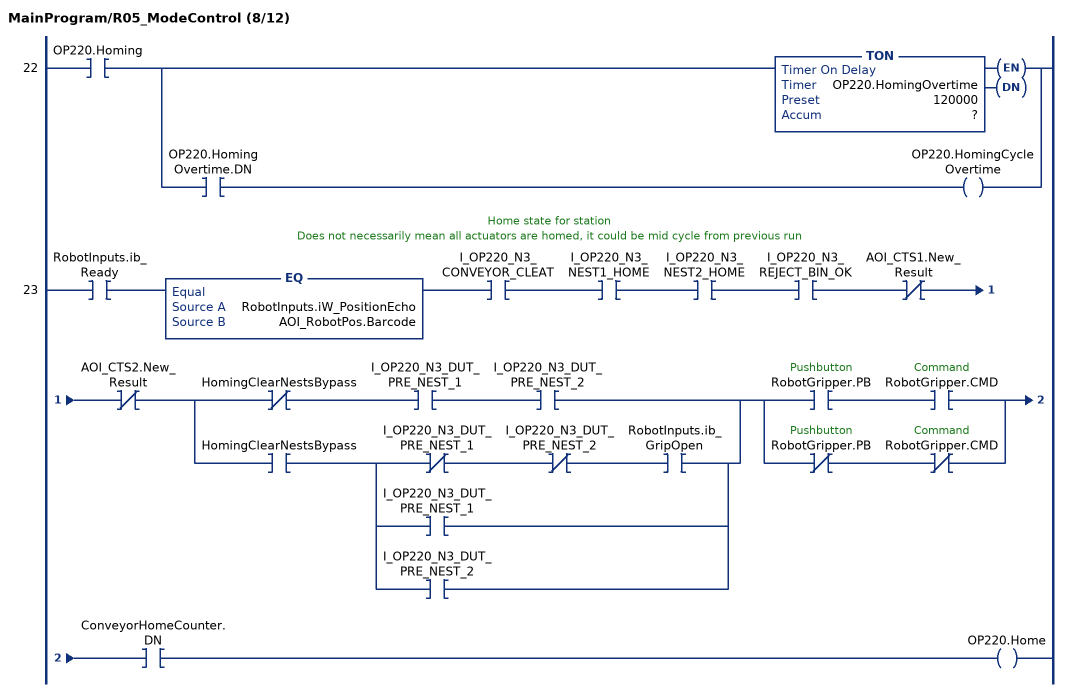
   22: XIC(OP220.Homing)[TON(OP220.HomingOvertime,?,?) ,XIC(OP220.HomingOvertime.DN) OTE(OP220.HomingCycleOvertime) ];
   // Home state for station
   // Does not necessarily mean all actuators are homed, it could be mid cycle from previous run
   23: XIC(RobotInputs.ib_Ready)EQ(RobotInputs.iW_PositionEcho,AOI_RobotPos.Barcode)XIC(I_OP220_N3_CONVEYOR_CLEAT)XIC(I_OP220_N3_NEST1_HOME)XIC(I_OP220_N3_NEST2_HOME)XIC(I_OP220_N3_REJECT_BIN_OK)XIO(AOI_CTS1.New_Result)XIO(AOI_CTS2.New_Result)[XIO(HomingClearNestsBypass) XIC(I_OP220_N3_DUT_PRE_NEST_1) XIC(I_OP220_N3_DUT_PRE_NEST_2) ,XIC(HomingClearNestsBypass) [XIO(I_OP220_N3_DUT_PRE_NEST_1) XIO(I_OP220_N3_DUT_PRE_NEST_2) XIC(RobotInputs.ib_GripOpen) ,XIC(I_OP220_N3_DUT_PRE_NEST_1) ,XIC(I_OP220_N3_DUT_PRE_NEST_2) ] ][XIC(RobotGripper.PB) XIC(RobotGripper.CMD) ,XIO(RobotGripper.PB) XIO(RobotGripper.CMD) ]XIC(ConveyorHomeCounter.DN)OTE(OP220.Home);
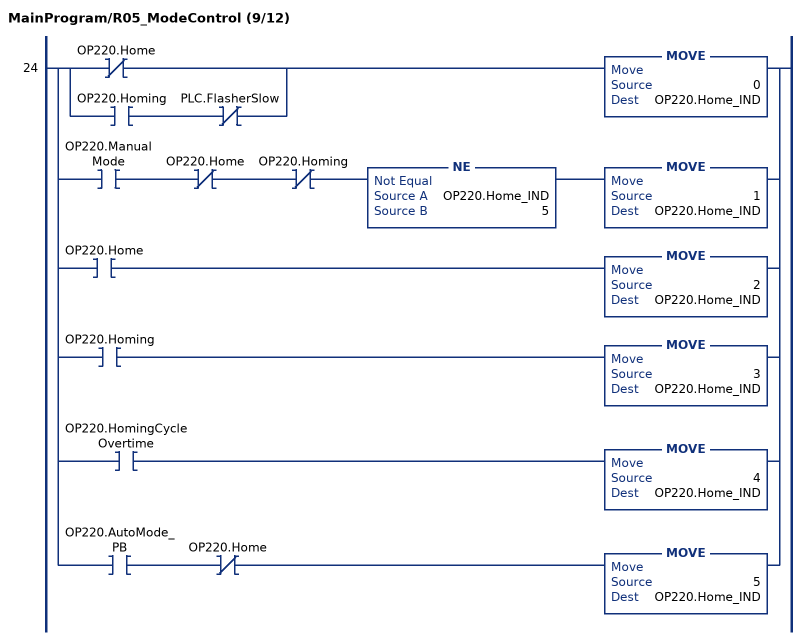
   24: [[XIO(OP220.Home) ,XIC(OP220.Homing) XIO(PLC.FlasherSlow) ] MOVE(0,OP220.Home_IND) ,XIC(OP220.ManualMode) XIO(OP220.Home) XIO(OP220.Homing) NE(OP220.Home_IND,5) MOVE(1,OP220.Home_IND) ,XIC(OP220.Home) MOVE(2,OP220.Home_IND) ,XIC(OP220.Homing) MOVE(3,OP220.Home_IND) ,XIC(OP220.HomingCycleOvertime) MOVE(4,OP220.Home_IND) ,XIC(OP220.AutoMode_PB) XIO(OP220.Home) MOVE(5,OP220.Home_IND) ];
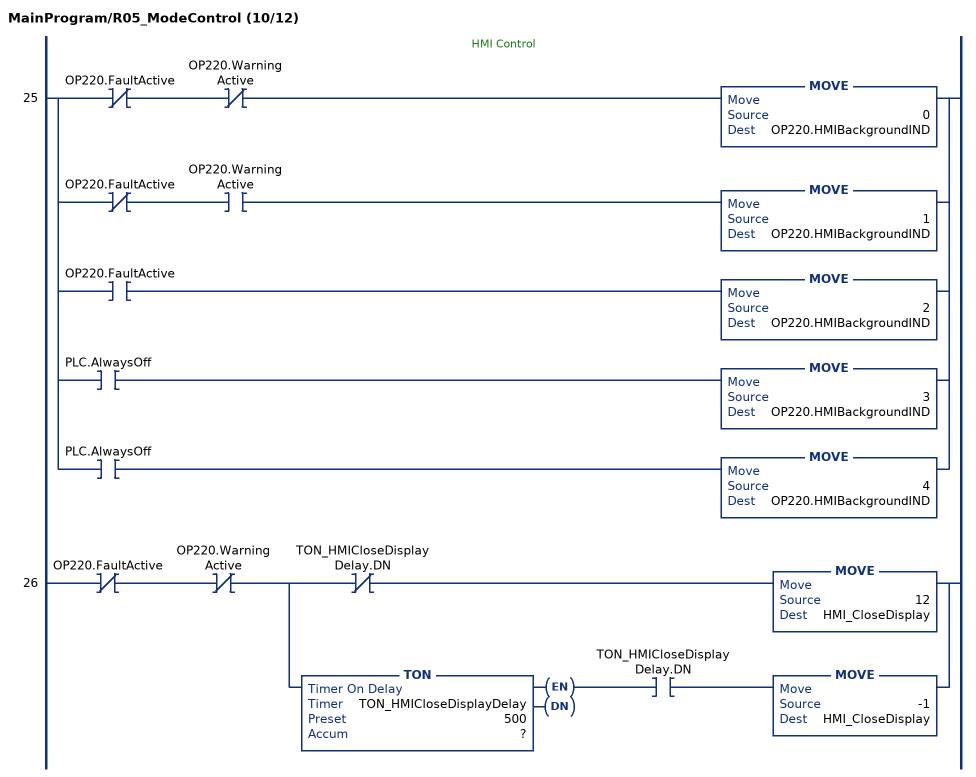
   // HMI Control
   25: [XIO(OP220.FaultActive) XIO(OP220.WarningActive) MOVE(0,OP220.HMIBackgroundIND) ,XIO(OP220.FaultActive) XIC(OP220.WarningActive) MOVE(1,OP220.HMIBackgroundIND) ,XIC(OP220.FaultActive) MOVE(2,OP220.HMIBackgroundIND) ,XIC(PLC.AlwaysOff) MOVE(3,OP220.HMIBackgroundIND) ,XIC(PLC.AlwaysOff) MOVE(4,OP220.HMIBackgroundIND) ];
   26: XIO(OP220.FaultActive)XIO(OP220.WarningActive)[XIO(TON_HMICloseDisplayDelay.DN) MOVE(12,HMI_CloseDisplay) ,TON(TON_HMICloseDisplayDelay,?,?) XIC(TON_HMICloseDisplayDelay.DN) MOVE(-1,HMI_CloseDisplay) ];
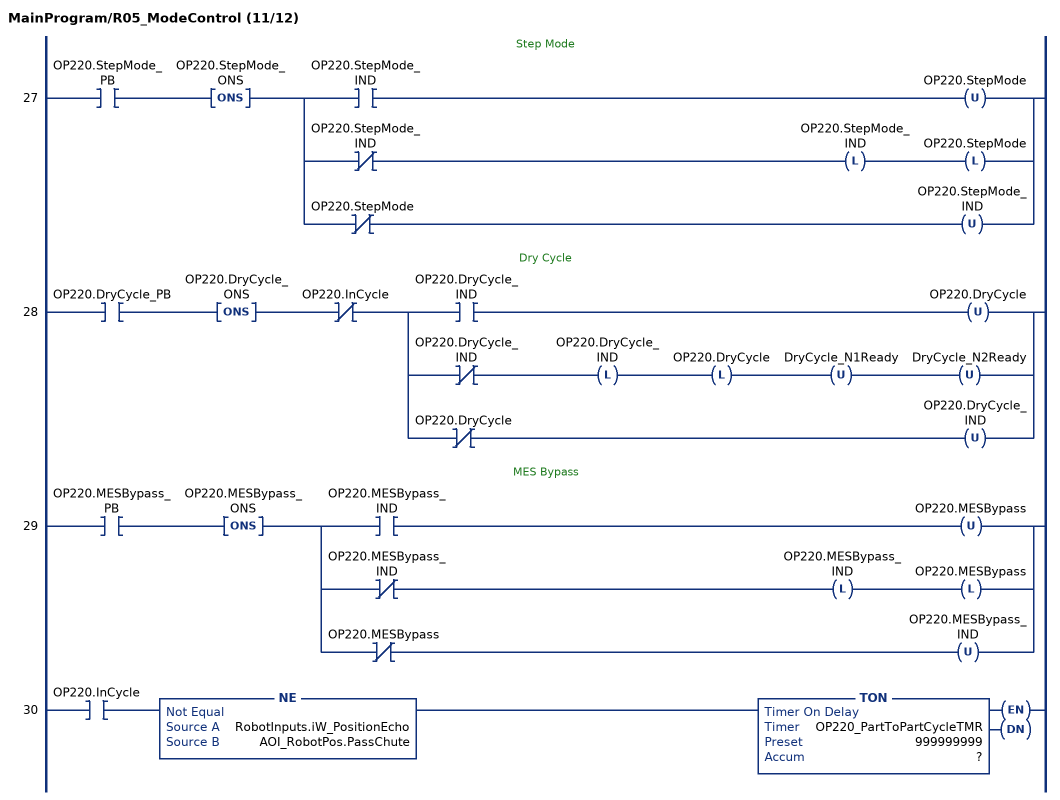
   // Step Mode
   27: XIC(OP220.StepMode_PB)ONS(OP220.StepMode_ONS)[XIC(OP220.StepMode_IND) OTU(OP220.StepMode) ,XIO(OP220.StepMode_IND) OTL(OP220.StepMode_IND) OTL(OP220.StepMode) ,XIO(OP220.StepMode) OTU(OP220.StepMode_IND) ];
   // Dry Cycle
   28: XIC(OP220.DryCycle_PB)ONS(OP220.DryCycle_ONS)XIO(OP220.InCycle)[XIC(OP220.DryCycle_IND) OTU(OP220.DryCycle) ,XIO(OP220.DryCycle_IND) OTL(OP220.DryCycle_IND) OTL(OP220.DryCycle) OTU(DryCycle_N1Ready) OTU(DryCycle_N2Ready) ,XIO(OP220.DryCycle) OTU(OP220.DryCycle_IND) ];
   // MES Bypass
   29: XIC(OP220.MESBypass_PB)ONS(OP220.MESBypass_ONS)[XIC(OP220.MESBypass_IND) OTU(OP220.MESBypass) ,XIO(OP220.MESBypass_IND) OTL(OP220.MESBypass_IND) OTL(OP220.MESBypass) ,XIO(OP220.MESBypass) OTU(OP220.MESBypass_IND) ];
   30: XIC(OP220.InCycle)NE(RobotInputs.iW_PositionEcho,AOI_RobotPos.PassChute)TON(OP220_PartToPartCycleTMR,?,?);
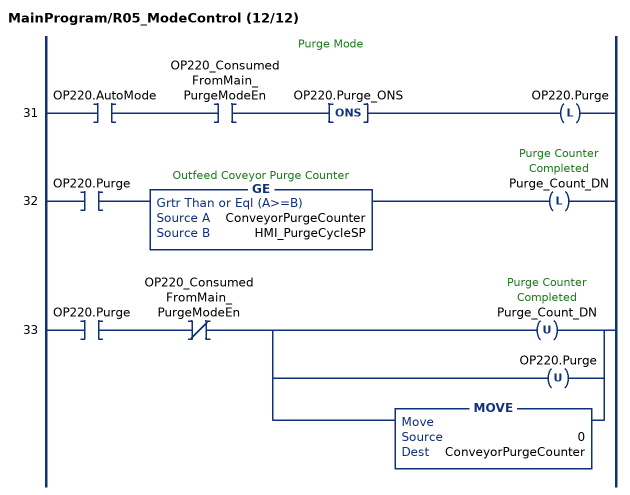
   // Purge Mode
   31: XIC(OP220.AutoMode)XIC(OP220_ConsumedFromMain_PurgeModeEn)ONS(OP220.Purge_ONS)OTL(OP220.Purge);
   32: XIC(OP220.Purge)GE(ConveyorPurgeCounter,HMI_PurgeCycleSP)OTL(Purge_Count_DN);
   33: XIC(OP220.Purge)XIO(OP220_ConsumedFromMain_PurgeModeEn)[OTU(Purge_Count_DN) ,OTU(OP220.Purge) ,MOVE(0,ConveyorPurgeCounter) ];
END_ROUTINE
